LIN {X 0,Y 584.166,Z 578.172,A -85,B 0,C 180,E1 27168.047,E2 27168.047} C_VEL
LIN {X 0,Y 584.179,Z 576.67,A -85,B 0,C 180,E1 27167.893,E2 27167.893} C_VEL
LIN {X 0,Y 583.247,Z 571.34,A -85,B 0,C 180,E1 27167.345,E2 27167.345} C_VEL
LIN {X 0,Y 577.743,Z 558.263,A -85,B 0,C 180,E1 27166.095,E2 27166.095} C_VEL
LIN {X 0,Y 576.592,Z 552.276,A -85,B 0,C 180,E1 27165.618,E2 27165.618} C_VEL
LIN {X 0,Y 576.579,Z 551.371,A -85,B 0,C 180,E1 27165.553,E2 27165.553} C_VEL
LIN {X 0,Y 576.766,Z 536.079,A -85,B 0,C 180,E1 27164.583,E2 27164.583} C_VEL
LIN {X 0,Y 576.943,Z 519.51,A -85,B 0,C 180,E1 27163.761,E2 27163.761} C_VEL
LIN {X 0,Y 577.114,Z 502.31,A -85,B 0,C 180,E1 27163.13,E2 27163.13} C_VEL
LIN {X 0,Y 577.241,Z 485.032,A -85,B 0,C 180,E1 27162.689,E2 27162.689} C_VEL
LIN {X 0,Y 577.308,Z 459.491,A -85,B 0,C 180,E1 27162.321,E2 27162.321} C_VEL
LIN {X 0,Y 577.408,Z 315.564,A -85,B 0,C 180,E1 27160.474,E2 27160.474} C_VEL
LIN {X 0,Y 576.956,Z 312.588,A -85,B 0,C 180,E1 27160.407,E2 27160.407} C_VEL
LIN {X 0,Y 577.293,Z 276.085,A -85,B 0,C 180,E1 27157.226,E2 27157.226} C_VEL
LIN {X 0,Y 577.599,Z 242.251,A -85,B 0,C 180,E1 27154.246,E2 27154.246} C_VEL
LIN {X 0,Y 577.82,Z 208.346,A -85,B 0,C 180,E1 27151.246,E2 27151.246} C_VEL
LIN {X 0,Y 577.684,Z 175.567,A -85,B 0,C 180,E1 27148.382,E2 27148.382} C_VEL
LIN {X 0,Y 576.141,Z 169.97,A -85,B 0,C 180,E1 27147.806,E2 27147.806} C_VEL
LIN {X 0,Y 576.151,Z 169.971,A -85,B 0,C 180,E1 27144.48,E2 27144.48} C_VEL
LIN {X 0,Y 576.179,Z 170.097,A -85,B 0,C 180,E1 27141.143,E2 27141.143} C_VEL
LIN {X 0,Y 577.537,Z 173.559,A -85,B 0,C 180,E1 27141,E2 27141} C_VEL
LIN {X 0,Y 580.966,Z 179.3,A -85,B 0,C 180,E1 27140.689,E2 27140.689} C_VEL
LIN {X 0,Y 580.065,Z 404.117,A -85,B 0,C 180,E1 27137.526,E2 27137.526} C_VEL
LIN {X 0,Y 579.833,Z 463.496,A -85,B 0,C 180,E1 27136.673,E2 27136.673} C_VEL
LIN {X 0,Y 579.571,Z 484.812,A -85,B 0,C 180,E1 27136.178,E2 27136.178} C_VEL
LIN {X 0,Y 579.218,Z 506.984,A -85,B 0,C 180,E1 27135.474,E2 27135.474} C_VEL
LIN {X 0,Y 578.916,Z 528.199,A -85,B 0,C 180,E1 27134.601,E2 27134.601} C_VEL
LIN {X 0,Y 578.485,Z 549.01,A -85,B 0,C 180,E1 27133.533,E2 27133.533} C_VEL
LIN {X 0,Y 578.045,Z 569.167,A -85,B 0,C 180,E1 27132.289,E2 27132.289} C_VEL
LIN {X 0,Y 577.637,Z 588.568,A -85,B 0,C 180,E1 27130.867,E2 27130.867} C_VEL
LIN {X 0,Y 577.271,Z 606.408,A -85,B 0,C 180,E1 27129.341,E2 27129.341} C_VEL
LIN {X 0,Y 576.911,Z 623.556,A -85,B 0,C 180,E1 27127.623,E2 27127.623} C_VEL
LIN {X 0,Y 576.612,Z 638.899,A -85,B 0,C 180,E1 27125.836,E2 27125.836} C_VEL
LIN {X 0,Y 576.369,Z 652.746,A -85,B 0,C 180,E1 27123.959,E2 27123.959} C_VEL
LIN {X 0,Y 576.211,Z 664.765,A -85,B 0,C 180,E1 27122.072,E2 27122.072} C_VEL
LIN {X 0,Y 576.076,Z 675.919,A -85,B 0,C 180,E1 27119.991,E2 27119.991} C_VEL
LIN {X 0,Y 575.987,Z 685.052,A -85,B 0,C 180,E1 27117.922,E2 27117.922} C_VEL
LIN {X 0,Y 575.944,Z 692.576,A -85,B 0,C 180,E1 27115.833,E2 27115.833} C_VEL
LIN {X 0,Y 575.929,Z 698.241,A -85,B 0,C 180,E1 27113.805,E2 27113.805} C_VEL
LIN {X 0,Y 575.915,Z 702.695,A -85,B 0,C 180,E1 27111.596,E2 27111.596} C_VEL
LIN {X 0,Y 575.902,Z 705.381,A -85,B 0,C 180,E1 27109.472,E2 27109.472} C_VEL
LIN {X 0,Y 575.902,Z 706.413,A -85,B 0,C 180,E1 27107.375,E2 27107.375} C_VEL
LIN {X 0,Y 575.913,Z 705.871,A -85,B 0,C 180,E1 27105.139,E2 27105.139} C_VEL
LIN {X 0,Y 575.912,Z 703.824,A -85,B 0,C 180,E1 27103.044,E2 27103.044} C_VEL
LIN {X 0,Y 575.916,Z 700.064,A -85,B 0,C 180,E1 27100.908,E2 27100.908} C_VEL
LIN {X 0,Y 575.928,Z 694.42,A -85,B 0,C 180,E1 27098.687,E2 27098.687} C_VEL
LIN {X 0,Y 575.978,Z 687.766,A -85,B 0,C 180,E1 27096.679,E2 27096.679} C_VEL
LIN {X 0,Y 576.046,Z 679.006,A -85,B 0,C 180,E1 27094.58,E2 27094.58} C_VEL
LIN {X 0,Y 576.161,Z 668.424,A -85,B 0,C 180,E1 27092.487,E2 27092.487} C_VEL
LIN {X 0,Y 576.33,Z 656.46,A -85,B 0,C 180,E1 27090.497,E2 27090.497} C_VEL
LIN {X 0,Y 576.542,Z 643.064,A -85,B 0,C 180,E1 27088.609,E2 27088.609} C_VEL
LIN {X 0,Y 576.8,Z 628.359,A -85,B 0,C 180,E1 27086.82,E2 27086.82} C_VEL
LIN {X 0,Y 577.132,Z 611.742,A -85,B 0,C 180,E1 27085.081,E2 27085.081} C_VEL
LIN {X 0,Y 577.525,Z 594.068,A -85,B 0,C 180,E1 27083.489,E2 27083.489} C_VEL
LIN {X 0,Y 577.918,Z 576.003,A -85,B 0,C 180,E1 27082.094,E2 27082.094} C_VEL
LIN {X 0,Y 578.324,Z 556.324,A -85,B 0,C 180,E1 27080.803,E2 27080.803} C_VEL
LIN {X 0,Y 578.737,Z 535.219,A -85,B 0,C 180,E1 27079.649,E2 27079.649} C_VEL
LIN {X 0,Y 579.132,Z 515.257,A -85,B 0,C 180,E1 27078.75,E2 27078.75} C_VEL
LIN {X 0,Y 579.447,Z 493.278,A -85,B 0,C 180,E1 27077.974,E2 27077.974} C_VEL
LIN {X 0,Y 579.733,Z 471.198,A -85,B 0,C 180,E1 27077.398,E2 27077.398} C_VEL
LIN {X 0,Y 579.913,Z 449.201,A -85,B 0,C 180,E1 27077.008,E2 27077.008} C_VEL
LIN {X 0,Y 580.632,Z 243.532,A -85,B 0,C 180,E1 27074.13,E2 27074.13} C_VEL
LIN {X 0,Y 580.771,Z 178.82,A -85,B 0,C 180,E1 27073.202,E2 27073.202} C_VEL
LIN {X 0,Y 576.397,Z 171.192,A -85,B 0,C 180,E1 27072.798,E2 27072.798} C_VEL
LIN {X 0,Y 576.14,Z 169.971,A -85,B 0,C 180,E1 27072.737,E2 27072.737} C_VEL
LIN {X 0,Y 576.15,Z 169.971,A -85,B 0,C 180,E1 27069.479,E2 27069.479} C_VEL
LIN {X 0,Y 576.138,Z 169.966,A -85,B 0,C 180,E1 27066.258,E2 27066.258} C_VEL
LIN {X 0,Y 576.153,Z 169.963,A -85,B 0,C 180,E1 27062.956,E2 27062.956} C_VEL
LIN {X 0,Y 576.12,Z 169.969,A -85,B 0,C 180,E1 27059.667,E2 27059.667} C_VEL
LIN {X 0,Y 576.138,Z 169.97,A -85,B 0,C 180,E1 27056.411,E2 27056.411} C_VEL
LIN {X 0,Y 576.129,Z 169.971,A -85,B 0,C 180,E1 27053.136,E2 27053.136} C_VEL
LIN {X 0,Y 576.113,Z 169.969,A -85,B 0,C 180,E1 27049.918,E2 27049.918} C_VEL
LIN {X 0,Y 576.152,Z 169.964,A -85,B 0,C 180,E1 27046.647,E2 27046.647} C_VEL
LIN {X 0,Y 576.143,Z 169.967,A -85,B 0,C 180,E1 27043.352,E2 27043.352} C_VEL
LIN {X 0,Y 576.158,Z 169.967,A -85,B 0,C 180,E1 27040.066,E2 27040.066} C_VEL
LIN {X 0,Y 576.159,Z 169.965,A -85,B 0,C 180,E1 27036.703,E2 27036.703} C_VEL
LIN {X 0,Y 576.092,Z 169.971,A -85,B 0,C 180,E1 27033.499,E2 27033.499} C_VEL
LIN {X 0,Y 576.113,Z 169.968,A -85,B 0,C 180,E1 27030.104,E2 27030.104} C_VEL
LIN {X 0,Y 576.158,Z 169.964,A -85,B 0,C 180,E1 27026.876,E2 27026.876} C_VEL
LIN {X 0,Y 576.157,Z 169.966,A -85,B 0,C 180,E1 27023.525,E2 27023.525} C_VEL
LIN {X 0,Y 576.157,Z 169.967,A -85,B 0,C 180,E1 27020.203,E2 27020.203} C_VEL
LIN {X 0,Y 576.124,Z 169.965,A -85,B 0,C 180,E1 27017.009,E2 27017.009} C_VEL
LIN {X 0,Y 576.092,Z 169.967,A -85,B 0,C 180,E1 27013.756,E2 27013.756} C_VEL
LIN {X 0,Y 576.157,Z 169.967,A -85,B 0,C 180,E1 27010.6,E2 27010.6} C_VEL
LIN {X 0,Y 576.133,Z 169.968,A -85,B 0,C 180,E1 27007.379,E2 27007.379} C_VEL
LIN {X 0,Y 576.14,Z 169.962,A -85,B 0,C 180,E1 27004.081,E2 27004.081} C_VEL
LIN {X 0,Y 576.14,Z 169.964,A -85,B 0,C 180,E1 27000.895,E2 27000.895} C_VEL
LIN {X 0,Y 576.124,Z 169.969,A -85,B 0,C 180,E1 26997.514,E2 26997.514} C_VEL
LIN {X 0,Y 576.157,Z 169.969,A -85,B 0,C 180,E1 26994.323,E2 26994.323} C_VEL
LIN {X 0,Y 576.104,Z 169.969,A -85,B 0,C 180,E1 26991.115,E2 26991.115} C_VEL
LIN {X 0,Y 576.118,Z 169.965,A -85,B 0,C 180,E1 26987.878,E2 26987.878} C_VEL
LIN {X 0,Y 576.155,Z 169.964,A -85,B 0,C 180,E1 26984.706,E2 26984.706} C_VEL
LIN {X 0,Y 576.155,Z 169.968,A -85,B 0,C 180,E1 26981.357,E2 26981.357} C_VEL
LIN {X 0,Y 576.158,Z 169.964,A -85,B 0,C 180,E1 26978.093,E2 26978.093} C_VEL
LIN {X 0,Y 576.11,Z 169.969,A -85,B 0,C 180,E1 26974.946,E2 26974.946} C_VEL
LIN {X 0,Y 576.091,Z 169.971,A -85,B 0,C 180,E1 26971.605,E2 26971.605} C_VEL
LIN {X 0,Y 576.164,Z 169.967,A -85,B 0,C 180,E1 26968.51,E2 26968.51} C_VEL
LIN {X 0,Y 576.144,Z 169.97,A -85,B 0,C 180,E1 26965.171,E2 26965.171} C_VEL
LIN {X 0,Y 576.163,Z 170.139,A -85,B 0,C 180,E1 26963.964,E2 26963.964} C_VEL
LIN {X 0,Y 577.514,Z 173.558,A -85,B 0,C 180,E1 26963.57,E2 26963.57} C_VEL
LIN {X 0,Y 581.885,Z 182.987,A -85,B 0,C 180,E1 26962.442,E2 26962.442} C_VEL
LIN {X 0,Y 581.171,Z 223.856,A -85,B 0,C 180,E1 26959.435,E2 26959.435} C_VEL
LIN {X 0,Y 580.968,Z 264.821,A -85,B 0,C 180,E1 26956.496,E2 26956.496} C_VEL
LIN {X 0,Y 582.558,Z 275.609,A -85,B 0,C 180,E1 26955.621,E2 26955.621} C_VEL
LIN {X 0,Y 585.556,Z 284.297,A -85,B 0,C 180,E1 26954.808,E2 26954.808} C_VEL
LIN {X 0,Y 589.359,Z 290.159,A -85,B 0,C 180,E1 26954.141,E2 26954.141} C_VEL
LIN {X 0,Y 592.357,Z 293.003,A -85,B 0,C 180,E1 26953.604,E2 26953.604} C_VEL
LIN {X 0,Y 594.862,Z 294.195,A -85,B 0,C 180,E1 26953.017,E2 26953.017} C_VEL
LIN {X 0,Y 596.402,Z 293.842,A -85,B 0,C 180,E1 26952.469,E2 26952.469} C_VEL
LIN {X 0,Y 597.06,Z 292.212,A -85,B 0,C 180,E1 26951.927,E2 26951.927} C_VEL
LIN {X 0,Y 596.652,Z 289.094,A -85,B 0,C 180,E1 26951.383,E2 26951.383} C_VEL
LIN {X 0,Y 595.08,Z 284.676,A -85,B 0,C 180,E1 26950.925,E2 26950.925} C_VEL
LIN {X 0,Y 592.307,Z 278.496,A -85,B 0,C 180,E1 26950.559,E2 26950.559} C_VEL
LIN {X 0,Y 589.472,Z 269.594,A -85,B 0,C 180,E1 26950.235,E2 26950.235} C_VEL
LIN {X 0,Y 587.68,Z 259.22,A -85,B 0,C 180,E1 26950.028,E2 26950.028} C_VEL
LIN {X 0,Y 586.902,Z 246.138,A -85,B 0,C 180,E1 26949.938,E2 26949.938} C_VEL
LIN {X 0,Y 586.776,Z 183.916,A -85,B 0,C 180,E1 26949.923,E2 26949.923} C_VEL
LIN {X 0,Y 584.935,Z 181.56,A -85,B 0,C 180,E1 26949.707,E2 26949.707} C_VEL
LIN {X 0,Y 581.754,Z 178.104,A -85,B 0,C 180,E1 26949.329,E2 26949.329} C_VEL
LIN {X 0,Y 580.647,Z 176.215,A -85,B 0,C 180,E1 26949.195,E2 26949.195} C_VEL
LIN {X 0,Y 577.814,Z 173.937,A -85,B 0,C 180,E1 26948.849,E2 26948.849} C_VEL
LIN {X 0,Y 576.366,Z 171.038,A -85,B 0,C 180,E1 26948.67,E2 26948.67} C_VEL
LIN {X 0,Y 576.158,Z 169.97,A -85,B 0,C 180,E1 26948.627,E2 26948.627} C_VEL
LIN {X 0,Y 576.181,Z 170.151,A -85,B 0,C 180,E1 26948.44,E2 26948.44} C_VEL
LIN {X 0,Y 580.511,Z 180.927,A -85,B 0,C 180,E1 26947.321,E2 26947.321} C_VEL
LIN {X 0,Y 579.808,Z 224.835,A -85,B 0,C 180,E1 26944.266,E2 26944.266} C_VEL
LIN {X 0,Y 579.906,Z 227.325,A -85,B 0,C 180,E1 26944.125,E2 26944.125} C_VEL
LIN {X 0,Y 581.019,Z 234.139,A -85,B 0,C 180,E1 26943.951,E2 26943.951} C_VEL
LIN {X 0,Y 580.152,Z 452.345,A -85,B 0,C 180,E1 26940.873,E2 26940.873} C_VEL
LIN {X 0,Y 579.832,Z 532.96,A -85,B 0,C 180,E1 26939.727,E2 26939.727} C_VEL
LIN {X 0,Y 579.577,Z 555.095,A -85,B 0,C 180,E1 26939.217,E2 26939.217} C_VEL
LIN {X 0,Y 579.228,Z 577.783,A -85,B 0,C 180,E1 26938.49,E2 26938.49} C_VEL
LIN {X 0,Y 578.897,Z 598.757,A -85,B 0,C 180,E1 26937.62,E2 26937.62} C_VEL
LIN {X 0,Y 578.49,Z 618.753,A -85,B 0,C 180,E1 26936.593,E2 26936.593} C_VEL
LIN {X 0,Y 578.045,Z 638.958,A -85,B 0,C 180,E1 26935.347,E2 26935.347} C_VEL
LIN {X 0,Y 577.659,Z 658.111,A -85,B 0,C 180,E1 26933.95,E2 26933.95} C_VEL
LIN {X 0,Y 577.271,Z 676.271,A -85,B 0,C 180,E1 26932.399,E2 26932.399} C_VEL
LIN {X 0,Y 576.911,Z 693.951,A -85,B 0,C 180,E1 26930.629,E2 26930.629} C_VEL
LIN {X 0,Y 576.602,Z 709.761,A -85,B 0,C 180,E1 26928.775,E2 26928.775} C_VEL
LIN {X 0,Y 576.363,Z 723.17,A -85,B 0,C 180,E1 26926.944,E2 26926.944} C_VEL
LIN {X 0,Y 576.192,Z 735.515,A -85,B 0,C 180,E1 26924.984,E2 26924.984} C_VEL
LIN {X 0,Y 576.073,Z 746.408,A -85,B 0,C 180,E1 26922.938,E2 26922.938} C_VEL
LIN {X 0,Y 575.986,Z 755.302,A -85,B 0,C 180,E1 26920.907,E2 26920.907} C_VEL
LIN {X 0,Y 575.938,Z 762.863,A -85,B 0,C 180,E1 26918.788,E2 26918.788} C_VEL
LIN {X 0,Y 575.925,Z 768.682,A -85,B 0,C 180,E1 26916.68,E2 26916.68} C_VEL
LIN {X 0,Y 575.916,Z 772.79,A -85,B 0,C 180,E1 26914.58,E2 26914.58} C_VEL
LIN {X 0,Y 575.91,Z 775.488,A -85,B 0,C 180,E1 26912.388,E2 26912.388} C_VEL
LIN {X 0,Y 575.905,Z 776.473,A -85,B 0,C 180,E1 26910.199,E2 26910.199} C_VEL
LIN {X 0,Y 575.909,Z 775.822,A -85,B 0,C 180,E1 26908.109,E2 26908.109} C_VEL
LIN {X 0,Y 575.913,Z 773.582,A -85,B 0,C 180,E1 26905.918,E2 26905.918} C_VEL
LIN {X 0,Y 575.917,Z 769.79,A -85,B 0,C 180,E1 26903.821,E2 26903.821} C_VEL
LIN {X 0,Y 575.934,Z 764.368,A -85,B 0,C 180,E1 26901.711,E2 26901.711} C_VEL
LIN {X 0,Y 575.976,Z 757.695,A -85,B 0,C 180,E1 26899.7,E2 26899.7} C_VEL
LIN {X 0,Y 576.042,Z 749.224,A -85,B 0,C 180,E1 26897.672,E2 26897.672} C_VEL
LIN {X 0,Y 576.161,Z 738.987,A -85,B 0,C 180,E1 26895.631,E2 26895.631} C_VEL
LIN {X 0,Y 576.325,Z 727.346,A -85,B 0,C 180,E1 26893.677,E2 26893.677} C_VEL
LIN {X 0,Y 576.52,Z 714.246,A -85,B 0,C 180,E1 26891.809,E2 26891.809} C_VEL
LIN {X 0,Y 576.788,Z 698.895,A -85,B 0,C 180,E1 26889.926,E2 26889.926} C_VEL
LIN {X 0,Y 577.124,Z 682.718,A -85,B 0,C 180,E1 26888.219,E2 26888.219} C_VEL
LIN {X 0,Y 577.506,Z 665.385,A -85,B 0,C 180,E1 26886.642,E2 26886.642} C_VEL
LIN {X 0,Y 577.903,Z 646.751,A -85,B 0,C 180,E1 26885.193,E2 26885.193} C_VEL
LIN {X 0,Y 578.302,Z 627.096,A -85,B 0,C 180,E1 26883.895,E2 26883.895} C_VEL
LIN {X 0,Y 578.73,Z 606.41,A -85,B 0,C 180,E1 26882.752,E2 26882.752} C_VEL
LIN {X 0,Y 579.124,Z 585.901,A -85,B 0,C 180,E1 26881.823,E2 26881.823} C_VEL
LIN {X 0,Y 579.425,Z 564.416,A -85,B 0,C 180,E1 26881.056,E2 26881.056} C_VEL
LIN {X 0,Y 579.735,Z 542.303,A -85,B 0,C 180,E1 26880.466,E2 26880.466} C_VEL
LIN {X 0,Y 579.913,Z 520.195,A -85,B 0,C 180,E1 26880.067,E2 26880.067} C_VEL
LIN {X 0,Y 580.782,Z 292.439,A -85,B 0,C 180,E1 26876.88,E2 26876.88} C_VEL
LIN {X 0,Y 580.844,Z 228.358,A -85,B 0,C 180,E1 26875.953,E2 26875.953} C_VEL
LIN {X 0,Y 580.391,Z 224.044,A -85,B 0,C 180,E1 26875.832,E2 26875.832} C_VEL
LIN {X 0,Y 580.924,Z 180.697,A -85,B 0,C 180,E1 26873.742,E2 26873.742} C_VEL
LIN {X 0,Y 576.27,Z 170.651,A -85,B 0,C 180,E1 26872.894,E2 26872.894} C_VEL
LIN {X 0,Y 576.152,Z 169.971,A -85,B 0,C 180,E1 26872.848,E2 26872.848} C_VEL
LIN {X 0,Y 576.184,Z 170.204,A -85,B 0,C 180,E1 26871.352,E2 26871.352} C_VEL
LIN {X 0,Y 577.268,Z 173.153,A -85,B 0,C 180,E1 26871.218,E2 26871.218} C_VEL
LIN {X 0,Y 579.702,Z 175.67,A -85,B 0,C 180,E1 26870.92,E2 26870.92} C_VEL
LIN {X 0,Y 580.965,Z 176.724,A -85,B 0,C 180,E1 26870.766,E2 26870.766} C_VEL
LIN {X 0,Y 583.703,Z 180.482,A -85,B 0,C 180,E1 26870.438,E2 26870.438} C_VEL
LIN {X 0,Y 585.977,Z 182.712,A -85,B 0,C 180,E1 26870.17,E2 26870.17} C_VEL
LIN {X 0,Y 589.596,Z 186.957,A -85,B 0,C 180,E1 26869.75,E2 26869.75} C_VEL
LIN {X 0,Y 594.761,Z 192.611,A -85,B 0,C 180,E1 26869.159,E2 26869.159} C_VEL
LIN {X 0,Y 597.542,Z 195.032,A -85,B 0,C 180,E1 26868.691,E2 26868.691} C_VEL
LIN {X 0,Y 599.27,Z 196.446,A -85,B 0,C 180,E1 26868.134,E2 26868.134} C_VEL
LIN {X 0,Y 599.686,Z 197.232,A -85,B 0,C 180,E1 26867.613,E2 26867.613} C_VEL
LIN {X 0,Y 598.696,Z 198.051,A -85,B 0,C 180,E1 26867.011,E2 26867.011} C_VEL
LIN {X 0,Y 596.915,Z 197.512,A -85,B 0,C 180,E1 26866.493,E2 26866.493} C_VEL
LIN {X 0,Y 594.088,Z 195.403,A -85,B 0,C 180,E1 26865.943,E2 26865.943} C_VEL
LIN {X 0,Y 591.068,Z 193.123,A -85,B 0,C 180,E1 26865.55,E2 26865.55} C_VEL
LIN {X 0,Y 585.889,Z 188.609,A -85,B 0,C 180,E1 26864.952,E2 26864.952} C_VEL
LIN {X 0,Y 582.45,Z 183.25,A -85,B 0,C 180,E1 26864.428,E2 26864.428} C_VEL
LIN {X 0,Y 576.337,Z 170.931,A -85,B 0,C 180,E1 26863.324,E2 26863.324} C_VEL
LIN {X 0,Y 576.158,Z 169.971,A -85,B 0,C 180,E1 26863.241,E2 26863.241} C_VEL
LIN {X 0,Y 576.139,Z 169.964,A -85,B 0,C 180,E1 26859.949,E2 26859.949} C_VEL
LIN {X 0,Y 576.118,Z 169.969,A -85,B 0,C 180,E1 26856.656,E2 26856.656} C_VEL
LIN {X 0,Y 576.161,Z 169.969,A -85,B 0,C 180,E1 26853.413,E2 26853.413} C_VEL
LIN {X 0,Y 576.162,Z 170.086,A -85,B 0,C 180,E1 26851.16,E2 26851.16} C_VEL
LIN {X 0,Y 576.697,Z 174.6,A -85,B 0,C 180,E1 26850.819,E2 26850.819} C_VEL
LIN {X 0,Y 577.409,Z 207.54,A -85,B 0,C 180,E1 26848.324,E2 26848.324} C_VEL
LIN {X 0,Y 577.599,Z 237.816,A -85,B 0,C 180,E1 26845.863,E2 26845.863} C_VEL
LIN {X 0,Y 577.369,Z 272.172,A -85,B 0,C 180,E1 26842.932,E2 26842.932} C_VEL
LIN {X 0,Y 576.978,Z 310.15,A -85,B 0,C 180,E1 26839.697,E2 26839.697} C_VEL
LIN {X 0,Y 576.997,Z 313.03,A -85,B 0,C 180,E1 26839.483,E2 26839.483} C_VEL
LIN {X 0,Y 577.561,Z 319.15,A -85,B 0,C 180,E1 26839.384,E2 26839.384} C_VEL
LIN {X 0,Y 577.209,Z 481.726,A -85,B 0,C 180,E1 26837.282,E2 26837.282} C_VEL
LIN {X 0,Y 577.127,Z 499.279,A -85,B 0,C 180,E1 26836.872,E2 26836.872} C_VEL
LIN {X 0,Y 576.991,Z 515.78,A -85,B 0,C 180,E1 26836.303,E2 26836.303} C_VEL
LIN {X 0,Y 576.811,Z 532.277,A -85,B 0,C 180,E1 26835.534,E2 26835.534} C_VEL
LIN {X 0,Y 576.635,Z 547.335,A -85,B 0,C 180,E1 26834.636,E2 26834.636} C_VEL
LIN {X 0,Y 576.449,Z 562.025,A -85,B 0,C 180,E1 26833.542,E2 26833.542} C_VEL
LIN {X 0,Y 576.281,Z 575.839,A -85,B 0,C 180,E1 26832.271,E2 26832.271} C_VEL
LIN {X 0,Y 576.151,Z 587.921,A -85,B 0,C 180,E1 26830.903,E2 26830.903} C_VEL
LIN {X 0,Y 576.044,Z 598.713,A -85,B 0,C 180,E1 26829.39,E2 26829.39} C_VEL
LIN {X 0,Y 575.978,Z 607.856,A -85,B 0,C 180,E1 26827.782,E2 26827.782} C_VEL
LIN {X 0,Y 575.941,Z 614.944,A -85,B 0,C 180,E1 26826.179,E2 26826.179} C_VEL
LIN {X 0,Y 575.924,Z 620.472,A -85,B 0,C 180,E1 26824.48,E2 26824.48} C_VEL
LIN {X 0,Y 575.915,Z 624.302,A -85,B 0,C 180,E1 26822.686,E2 26822.686} C_VEL
LIN {X 0,Y 575.909,Z 626.225,A -85,B 0,C 180,E1 26820.895,E2 26820.895} C_VEL
LIN {X 0,Y 575.914,Z 626.333,A -85,B 0,C 180,E1 26819.204,E2 26819.204} C_VEL
LIN {X 0,Y 575.915,Z 624.602,A -85,B 0,C 180,E1 26817.412,E2 26817.412} C_VEL
LIN {X 0,Y 575.921,Z 620.948,A -85,B 0,C 180,E1 26815.619,E2 26815.619} C_VEL
LIN {X 0,Y 575.935,Z 615.645,A -85,B 0,C 180,E1 26813.921,E2 26813.921} C_VEL
LIN {X 0,Y 575.976,Z 608.813,A -85,B 0,C 180,E1 26812.318,E2 26812.318} C_VEL
LIN {X 0,Y 576.035,Z 599.922,A -85,B 0,C 180,E1 26810.71,E2 26810.71} C_VEL
LIN {X 0,Y 576.13,Z 589.382,A -85,B 0,C 180,E1 26809.197,E2 26809.197} C_VEL
LIN {X 0,Y 576.266,Z 577.477,A -85,B 0,C 180,E1 26807.809,E2 26807.809} C_VEL
LIN {X 0,Y 576.418,Z 564.288,A -85,B 0,C 180,E1 26806.559,E2 26806.559} C_VEL
LIN {X 0,Y 576.579,Z 551.371,A -85,B 0,C 180,E1 26805.553,E2 26805.553} C_VEL
LIN {X 0,Y 575.681,Z 545.123,A -85,B 0,C 180,E1 26805.102,E2 26805.102} C_VEL
LIN {X 0,Y 570.3,Z 530.053,A -85,B 0,C 180,E1 26804.075,E2 26804.075} C_VEL
LIN {X 0,Y 569.181,Z 522.294,A -85,B 0,C 180,E1 26803.662,E2 26803.662} C_VEL
LIN {X 0,Y 569.387,Z 506.325,A -85,B 0,C 180,E1 26803.026,E2 26803.026} C_VEL
LIN {X 0,Y 569.555,Z 489.29,A -85,B 0,C 180,E1 26802.544,E2 26802.544} C_VEL
LIN {X 0,Y 569.665,Z 470.385,A -85,B 0,C 180,E1 26802.217,E2 26802.217} C_VEL
LIN {X 0,Y 569.852,Z 316.495,A -85,B 0,C 180,E1 26800.217,E2 26800.217} C_VEL
LIN {X 0,Y 569.247,Z 312.464,A -85,B 0,C 180,E1 26800.12,E2 26800.12} C_VEL
LIN {X 0,Y 569.705,Z 277.5,A -85,B 0,C 180,E1 26797.014,E2 26797.014} C_VEL
LIN {X 0,Y 570.079,Z 241.888,A -85,B 0,C 180,E1 26793.851,E2 26793.851} C_VEL
LIN {X 0,Y 570.312,Z 209.094,A -85,B 0,C 180,E1 26790.946,E2 26790.946} C_VEL
LIN {X 0,Y 570.279,Z 178.323,A -85,B 0,C 180,E1 26788.249,E2 26788.249} C_VEL
LIN {X 0,Y 568.213,Z 170.957,A -85,B 0,C 180,E1 26787.491,E2 26787.491} C_VEL
LIN {X 0,Y 568.193,Z 170.959,A -85,B 0,C 180,E1 26784.127,E2 26784.127} C_VEL
LIN {X 0,Y 568.211,Z 171.117,A -85,B 0,C 180,E1 26781.675,E2 26781.675} C_VEL
LIN {X 0,Y 569.487,Z 174.414,A -85,B 0,C 180,E1 26781.537,E2 26781.537} C_VEL
LIN {X 0,Y 571.236,Z 177.159,A -85,B 0,C 180,E1 26781.375,E2 26781.375} C_VEL
LIN {X 0,Y 574.293,Z 182.62,A -85,B 0,C 180,E1 26781.085,E2 26781.085} C_VEL
LIN {X 0,Y 573.165,Z 406.563,A -85,B 0,C 180,E1 26777.899,E2 26777.899} C_VEL
LIN {X 0,Y 572.876,Z 463.7,A -85,B 0,C 180,E1 26777.067,E2 26777.067} C_VEL
LIN {X 0,Y 572.549,Z 485.027,A -85,B 0,C 180,E1 26776.566,E2 26776.566} C_VEL
LIN {X 0,Y 572.135,Z 506.682,A -85,B 0,C 180,E1 26775.872,E2 26775.872} C_VEL
LIN {X 0,Y 571.735,Z 527.721,A -85,B 0,C 180,E1 26775.001,E2 26775.001} C_VEL
LIN {X 0,Y 571.185,Z 548.622,A -85,B 0,C 180,E1 26773.922,E2 26773.922} C_VEL
LIN {X 0,Y 570.668,Z 568.42,A -85,B 0,C 180,E1 26772.692,E2 26772.692} C_VEL
LIN {X 0,Y 570.164,Z 587.116,A -85,B 0,C 180,E1 26771.319,E2 26771.319} C_VEL
LIN {X 0,Y 569.683,Z 604.411,A -85,B 0,C 180,E1 26769.838,E2 26769.838} C_VEL
LIN {X 0,Y 569.224,Z 621.861,A -85,B 0,C 180,E1 26768.1,E2 26768.1} C_VEL
LIN {X 0,Y 568.85,Z 637.152,A -85,B 0,C 180,E1 26766.324,E2 26766.324} C_VEL
LIN {X 0,Y 568.536,Z 652.019,A -85,B 0,C 180,E1 26764.309,E2 26764.309} C_VEL
LIN {X 0,Y 568.321,Z 664.211,A -85,B 0,C 180,E1 26762.384,E2 26762.384} C_VEL
LIN {X 0,Y 568.134,Z 675.718,A -85,B 0,C 180,E1 26760.218,E2 26760.218} C_VEL
LIN {X 0,Y 568.021,Z 684.855,A -85,B 0,C 180,E1 26758.128,E2 26758.128} C_VEL
LIN {X 0,Y 567.963,Z 692.456,A -85,B 0,C 180,E1 26755.999,E2 26755.999} C_VEL
LIN {X 0,Y 567.933,Z 698.282,A -85,B 0,C 180,E1 26753.886,E2 26753.886} C_VEL
LIN {X 0,Y 567.914,Z 702.641,A -85,B 0,C 180,E1 26751.699,E2 26751.699} C_VEL
LIN {X 0,Y 567.901,Z 705.349,A -85,B 0,C 180,E1 26749.543,E2 26749.543} C_VEL
LIN {X 0,Y 567.902,Z 706.41,A -85,B 0,C 180,E1 26747.396,E2 26747.396} C_VEL
LIN {X 0,Y 567.915,Z 705.866,A -85,B 0,C 180,E1 26745.104,E2 26745.104} C_VEL
LIN {X 0,Y 567.91,Z 703.73,A -85,B 0,C 180,E1 26742.921,E2 26742.921} C_VEL
LIN {X 0,Y 567.911,Z 699.931,A -85,B 0,C 180,E1 26740.756,E2 26740.756} C_VEL
LIN {X 0,Y 567.934,Z 694.528,A -85,B 0,C 180,E1 26738.606,E2 26738.606} C_VEL
LIN {X 0,Y 567.993,Z 687.895,A -85,B 0,C 180,E1 26736.57,E2 26736.57} C_VEL
LIN {X 0,Y 568.081,Z 679.181,A -85,B 0,C 180,E1 26734.442,E2 26734.442} C_VEL
LIN {X 0,Y 568.226,Z 668.647,A -85,B 0,C 180,E1 26732.32,E2 26732.32} C_VEL
LIN {X 0,Y 568.441,Z 656.726,A -85,B 0,C 180,E1 26730.303,E2 26730.303} C_VEL
LIN {X 0,Y 568.716,Z 643.363,A -85,B 0,C 180,E1 26728.388,E2 26728.388} C_VEL
LIN {X 0,Y 569.054,Z 628.72,A -85,B 0,C 180,E1 26726.575,E2 26726.575} C_VEL
LIN {X 0,Y 569.476,Z 612.164,A -85,B 0,C 180,E1 26724.812,E2 26724.812} C_VEL
LIN {X 0,Y 569.949,Z 595.181,A -85,B 0,C 180,E1 26723.25,E2 26723.25} C_VEL
LIN {X 0,Y 570.447,Z 576.852,A -85,B 0,C 180,E1 26721.81,E2 26721.81} C_VEL
LIN {X 0,Y 570.951,Z 557.704,A -85,B 0,C 180,E1 26720.525,E2 26720.525} C_VEL
LIN {X 0,Y 571.458,Z 537.985,A -85,B 0,C 180,E1 26719.414,E2 26719.414} C_VEL
LIN {X 0,Y 571.899,Z 518.451,A -85,B 0,C 180,E1 26718.504,E2 26718.504} C_VEL
LIN {X 0,Y 572.34,Z 496.753,A -85,B 0,C 180,E1 26717.694,E2 26717.694} C_VEL
LIN {X 0,Y 572.729,Z 474.998,A -85,B 0,C 180,E1 26717.085,E2 26717.085} C_VEL
LIN {X 0,Y 572.93,Z 453.631,A -85,B 0,C 180,E1 26716.675,E2 26716.675} C_VEL
LIN {X 0,Y 573.884,Z 247.929,A -85,B 0,C 180,E1 26713.759,E2 26713.759} C_VEL
LIN {X 0,Y 574.094,Z 182.048,A -85,B 0,C 180,E1 26712.803,E2 26712.803} C_VEL
LIN {X 0,Y 569.856,Z 174.958,A -85,B 0,C 180,E1 26712.407,E2 26712.407} C_VEL
LIN {X 0,Y 568.271,Z 171.594,A -85,B 0,C 180,E1 26712.246,E2 26712.246} C_VEL
LIN {X 0,Y 568.165,Z 170.961,A -85,B 0,C 180,E1 26712.217,E2 26712.217} C_VEL
LIN {X 0,Y 568.223,Z 170.956,A -85,B 0,C 180,E1 26709.072,E2 26709.072} C_VEL
LIN {X 0,Y 568.218,Z 170.959,A -85,B 0,C 180,E1 26705.685,E2 26705.685} C_VEL
LIN {X 0,Y 568.216,Z 170.957,A -85,B 0,C 180,E1 26702.319,E2 26702.319} C_VEL
LIN {X 0,Y 568.197,Z 170.956,A -85,B 0,C 180,E1 26699.081,E2 26699.081} C_VEL
LIN {X 0,Y 568.156,Z 170.958,A -85,B 0,C 180,E1 26695.805,E2 26695.805} C_VEL
LIN {X 0,Y 568.189,Z 170.955,A -85,B 0,C 180,E1 26692.528,E2 26692.528} C_VEL
LIN {X 0,Y 568.215,Z 170.959,A -85,B 0,C 180,E1 26689.325,E2 26689.325} C_VEL
LIN {X 0,Y 568.198,Z 170.957,A -85,B 0,C 180,E1 26686.032,E2 26686.032} C_VEL
LIN {X 0,Y 568.217,Z 170.952,A -85,B 0,C 180,E1 26682.646,E2 26682.646} C_VEL
LIN {X 0,Y 568.183,Z 170.956,A -85,B 0,C 180,E1 26679.418,E2 26679.418} C_VEL
LIN {X 0,Y 568.185,Z 170.958,A -85,B 0,C 180,E1 26676.123,E2 26676.123} C_VEL
LIN {X 0,Y 568.199,Z 170.96,A -85,B 0,C 180,E1 26672.926,E2 26672.926} C_VEL
LIN {X 0,Y 568.171,Z 170.958,A -85,B 0,C 180,E1 26669.753,E2 26669.753} C_VEL
LIN {X 0,Y 568.214,Z 170.951,A -85,B 0,C 180,E1 26666.549,E2 26666.549} C_VEL
LIN {X 0,Y 568.205,Z 170.951,A -85,B 0,C 180,E1 26663.215,E2 26663.215} C_VEL
LIN {X 0,Y 568.217,Z 170.959,A -85,B 0,C 180,E1 26659.961,E2 26659.961} C_VEL
LIN {X 0,Y 568.212,Z 170.953,A -85,B 0,C 180,E1 26656.668,E2 26656.668} C_VEL
LIN {X 0,Y 568.149,Z 170.956,A -85,B 0,C 180,E1 26653.537,E2 26653.537} C_VEL
LIN {X 0,Y 568.197,Z 170.955,A -85,B 0,C 180,E1 26650.34,E2 26650.34} C_VEL
LIN {X 0,Y 568.225,Z 170.958,A -85,B 0,C 180,E1 26647.057,E2 26647.057} C_VEL
LIN {X 0,Y 568.207,Z 170.953,A -85,B 0,C 180,E1 26643.733,E2 26643.733} C_VEL
LIN {X 0,Y 568.22,Z 170.951,A -85,B 0,C 180,E1 26640.404,E2 26640.404} C_VEL
LIN {X 0,Y 568.177,Z 170.956,A -85,B 0,C 180,E1 26637.176,E2 26637.176} C_VEL
LIN {X 0,Y 568.171,Z 170.96,A -85,B 0,C 180,E1 26633.868,E2 26633.868} C_VEL
LIN {X 0,Y 568.21,Z 170.958,A -85,B 0,C 180,E1 26630.684,E2 26630.684} C_VEL
LIN {X 0,Y 568.186,Z 170.956,A -85,B 0,C 180,E1 26627.397,E2 26627.397} C_VEL
LIN {X 0,Y 568.202,Z 170.953,A -85,B 0,C 180,E1 26624.067,E2 26624.067} C_VEL
LIN {X 0,Y 568.203,Z 170.955,A -85,B 0,C 180,E1 26620.789,E2 26620.789} C_VEL
LIN {X 0,Y 568.192,Z 170.959,A -85,B 0,C 180,E1 26617.442,E2 26617.442} C_VEL
LIN {X 0,Y 568.223,Z 170.959,A -85,B 0,C 180,E1 26614.239,E2 26614.239} C_VEL
LIN {X 0,Y 568.167,Z 170.96,A -85,B 0,C 180,E1 26610.942,E2 26610.942} C_VEL
LIN {X 0,Y 568.175,Z 170.961,A -85,B 0,C 180,E1 26607.639,E2 26607.639} C_VEL
LIN {X 0,Y 568.218,Z 170.964,A -85,B 0,C 180,E1 26604.66,E2 26604.66} C_VEL
LIN {X 0,Y 569.643,Z 174.611,A -85,B 0,C 180,E1 26604.233,E2 26604.233} C_VEL
LIN {X 0,Y 575.394,Z 186.846,A -85,B 0,C 180,E1 26602.737,E2 26602.737} C_VEL
LIN {X 0,Y 574.517,Z 227.602,A -85,B 0,C 180,E1 26599.713,E2 26599.713} C_VEL
LIN {X 0,Y 574.164,Z 267.554,A -85,B 0,C 180,E1 26596.814,E2 26596.814} C_VEL
LIN {X 0,Y 575.799,Z 279.097,A -85,B 0,C 180,E1 26595.867,E2 26595.867} C_VEL
LIN {X 0,Y 578.917,Z 288.411,A -85,B 0,C 180,E1 26594.988,E2 26594.988} C_VEL
LIN {X 0,Y 582.683,Z 294.598,A -85,B 0,C 180,E1 26594.298,E2 26594.298} C_VEL
LIN {X 0,Y 587.242,Z 299.166,A -85,B 0,C 180,E1 26593.646,E2 26593.646} C_VEL
LIN {X 0,Y 590.318,Z 300.962,A -85,B 0,C 180,E1 26593.113,E2 26593.113} C_VEL
LIN {X 0,Y 592.765,Z 301.296,A -85,B 0,C 180,E1 26592.514,E2 26592.514} C_VEL
LIN {X 0,Y 594.139,Z 300.148,A -85,B 0,C 180,E1 26591.92,E2 26591.92} C_VEL
LIN {X 0,Y 594.316,Z 297.612,A -85,B 0,C 180,E1 26591.331,E2 26591.331} C_VEL
LIN {X 0,Y 593.247,Z 293.902,A -85,B 0,C 180,E1 26590.822,E2 26590.822} C_VEL
LIN {X 0,Y 591.037,Z 289.251,A -85,B 0,C 180,E1 26590.417,E2 26590.417} C_VEL
LIN {X 0,Y 587.259,Z 281.029,A -85,B 0,C 180,E1 26589.979,E2 26589.979} C_VEL
LIN {X 0,Y 584.417,Z 271.352,A -85,B 0,C 180,E1 26589.646,E2 26589.646} C_VEL
LIN {X 0,Y 582.587,Z 260.103,A -85,B 0,C 180,E1 26589.428,E2 26589.428} C_VEL
LIN {X 0,Y 581.802,Z 246.434,A -85,B 0,C 180,E1 26589.334,E2 26589.334} C_VEL
LIN {X 0,Y 581.754,Z 187.971,A -85,B 0,C 180,E1 26589.329,E2 26589.329} C_VEL
LIN {X 0,Y 578.128,Z 183.671,A -85,B 0,C 180,E1 26588.888,E2 26588.888} C_VEL
LIN {X 0,Y 574.536,Z 180.188,A -85,B 0,C 180,E1 26588.442,E2 26588.442} C_VEL
LIN {X 0,Y 572.522,Z 180.259,A -85,B 0,C 180,E1 26588.187,E2 26588.187} C_VEL
LIN {X 0,Y 571.743,Z 179.782,A -85,B 0,C 180,E1 26588.078,E2 26588.078} C_VEL
LIN {X 0,Y 573.683,Z 184.371,A -85,B 0,C 180,E1 26587.59,E2 26587.59} C_VEL
LIN {X 0,Y 572.909,Z 227.019,A -85,B 0,C 180,E1 26584.605,E2 26584.605} C_VEL
LIN {X 0,Y 574.375,Z 235.64,A -85,B 0,C 180,E1 26584.376,E2 26584.376} C_VEL
LIN {X 0,Y 573.274,Z 454.189,A -85,B 0,C 180,E1 26581.259,E2 26581.259} C_VEL
LIN {X 0,Y 572.877,Z 532.947,A -85,B 0,C 180,E1 26580.125,E2 26580.125} C_VEL
LIN {X 0,Y 572.556,Z 555.224,A -85,B 0,C 180,E1 26579.608,E2 26579.608} C_VEL
LIN {X 0,Y 572.139,Z 577.376,A -85,B 0,C 180,E1 26578.892,E2 26578.892} C_VEL
LIN {X 0,Y 571.707,Z 598.694,A -85,B 0,C 180,E1 26578.001,E2 26578.001} C_VEL
LIN {X 0,Y 571.187,Z 618.761,A -85,B 0,C 180,E1 26576.961,E2 26576.961} C_VEL
LIN {X 0,Y 570.673,Z 638.161,A -85,B 0,C 180,E1 26575.754,E2 26575.754} C_VEL
LIN {X 0,Y 570.182,Z 656.802,A -85,B 0,C 180,E1 26574.391,E2 26574.391} C_VEL
LIN {X 0,Y 569.662,Z 675.694,A -85,B 0,C 180,E1 26572.769,E2 26572.769} C_VEL
LIN {X 0,Y 569.199,Z 692.732,A -85,B 0,C 180,E1 26571.053,E2 26571.053} C_VEL
LIN {X 0,Y 568.838,Z 707.829,A -85,B 0,C 180,E1 26569.284,E2 26569.284} C_VEL
LIN {X 0,Y 568.545,Z 721.759,A -85,B 0,C 180,E1 26567.395,E2 26567.395} C_VEL
LIN {X 0,Y 568.31,Z 734.412,A -85,B 0,C 180,E1 26565.394,E2 26565.394} C_VEL
LIN {X 0,Y 568.139,Z 745.381,A -85,B 0,C 180,E1 26563.329,E2 26563.329} C_VEL
LIN {X 0,Y 568.022,Z 754.898,A -85,B 0,C 180,E1 26561.164,E2 26561.164} C_VEL
LIN {X 0,Y 567.965,Z 762.563,A -85,B 0,C 180,E1 26559.014,E2 26559.014} C_VEL
LIN {X 0,Y 567.933,Z 768.577,A -85,B 0,C 180,E1 26556.817,E2 26556.817} C_VEL
LIN {X 0,Y 567.918,Z 772.793,A -85,B 0,C 180,E1 26554.645,E2 26554.645} C_VEL
LIN {X 0,Y 567.909,Z 775.489,A -85,B 0,C 180,E1 26552.422,E2 26552.422} C_VEL
LIN {X 0,Y 567.905,Z 776.475,A -85,B 0,C 180,E1 26550.202,E2 26550.202} C_VEL
LIN {X 0,Y 567.912,Z 775.758,A -85,B 0,C 180,E1 26547.982,E2 26547.982} C_VEL
LIN {X 0,Y 567.911,Z 773.427,A -85,B 0,C 180,E1 26545.759,E2 26545.759} C_VEL
LIN {X 0,Y 567.916,Z 769.586,A -85,B 0,C 180,E1 26543.632,E2 26543.632} C_VEL
LIN {X 0,Y 567.936,Z 764.08,A -85,B 0,C 180,E1 26541.496,E2 26541.496} C_VEL
LIN {X 0,Y 567.995,Z 756.926,A -85,B 0,C 180,E1 26539.348,E2 26539.348} C_VEL
LIN {X 0,Y 568.088,Z 748.302,A -85,B 0,C 180,E1 26537.29,E2 26537.29} C_VEL
LIN {X 0,Y 568.231,Z 737.833,A -85,B 0,C 180,E1 26535.218,E2 26535.218} C_VEL
LIN {X 0,Y 568.452,Z 725.998,A -85,B 0,C 180,E1 26533.234,E2 26533.234} C_VEL
LIN {X 0,Y 568.756,Z 711.904,A -85,B 0,C 180,E1 26531.233,E2 26531.233} C_VEL
LIN {X 0,Y 569.105,Z 697.042,A -85,B 0,C 180,E1 26529.428,E2 26529.428} C_VEL
LIN {X 0,Y 569.526,Z 680.535,A -85,B 0,C 180,E1 26527.698,E2 26527.698} C_VEL
LIN {X 0,Y 569.996,Z 662.779,A -85,B 0,C 180,E1 26526.096,E2 26526.096} C_VEL
LIN {X 0,Y 570.521,Z 644.526,A -85,B 0,C 180,E1 26524.683,E2 26524.683} C_VEL
LIN {X 0,Y 571.061,Z 624.434,A -85,B 0,C 180,E1 26523.37,E2 26523.37} C_VEL
LIN {X 0,Y 571.529,Z 604.179,A -85,B 0,C 180,E1 26522.267,E2 26522.267} C_VEL
LIN {X 0,Y 572.047,Z 583.28,A -85,B 0,C 180,E1 26521.333,E2 26521.333} C_VEL
LIN {X 0,Y 572.454,Z 561.668,A -85,B 0,C 180,E1 26520.578,E2 26520.578} C_VEL
LIN {X 0,Y 572.77,Z 540.004,A -85,B 0,C 180,E1 26520.019,E2 26520.019} C_VEL
LIN {X 0,Y 573.001,Z 515.741,A -85,B 0,C 180,E1 26519.605,E2 26519.605} C_VEL
LIN {X 0,Y 574.094,Z 289.131,A -85,B 0,C 180,E1 26516.395,E2 26516.395} C_VEL
LIN {X 0,Y 574.203,Z 229.592,A -85,B 0,C 180,E1 26515.522,E2 26515.522} C_VEL
LIN {X 0,Y 573.604,Z 223.837,A -85,B 0,C 180,E1 26515.361,E2 26515.361} C_VEL
LIN {X 0,Y 574.113,Z 183.916,A -85,B 0,C 180,E1 26513.404,E2 26513.404} C_VEL
LIN {X 0,Y 569.318,Z 174.154,A -85,B 0,C 180,E1 26512.544,E2 26512.544} C_VEL
LIN {X 0,Y 568.414,Z 172.065,A -85,B 0,C 180,E1 26512.343,E2 26512.343} C_VEL
LIN {X 0,Y 569.906,Z 174.983,A -85,B 0,C 180,E1 26512.149,E2 26512.149} C_VEL
LIN {X 0,Y 572.832,Z 177.241,A -85,B 0,C 180,E1 26511.773,E2 26511.773} C_VEL
LIN {X 0,Y 575.783,Z 181.416,A -85,B 0,C 180,E1 26511.402,E2 26511.402} C_VEL
LIN {X 0,Y 578.208,Z 183.779,A -85,B 0,C 180,E1 26511.102,E2 26511.102} C_VEL
LIN {X 0,Y 581.756,Z 187.961,A -85,B 0,C 180,E1 26510.671,E2 26510.671} C_VEL
LIN {X 0,Y 591.863,Z 199.262,A -85,B 0,C 180,E1 26509.492,E2 26509.492} C_VEL
LIN {X 0,Y 594.914,Z 201.896,A -85,B 0,C 180,E1 26509.045,E2 26509.045} C_VEL
LIN {X 0,Y 596.981,Z 203.733,A -85,B 0,C 180,E1 26508.474,E2 26508.474} C_VEL
LIN {X 0,Y 597.659,Z 204.646,A -85,B 0,C 180,E1 26507.827,E2 26507.827} C_VEL
LIN {X 0,Y 596.61,Z 205.594,A -85,B 0,C 180,E1 26507.226,E2 26507.226} C_VEL
LIN {X 0,Y 594.296,Z 205.116,A -85,B 0,C 180,E1 26506.619,E2 26506.619} C_VEL
LIN {X 0,Y 591.192,Z 203.267,A -85,B 0,C 180,E1 26506.094,E2 26506.094} C_VEL
LIN {X 0,Y 586.722,Z 199.838,A -85,B 0,C 180,E1 26505.564,E2 26505.564} C_VEL
LIN {X 0,Y 581.489,Z 195.504,A -85,B 0,C 180,E1 26504.967,E2 26504.967} C_VEL
LIN {X 0,Y 577.456,Z 190.033,A -85,B 0,C 180,E1 26504.388,E2 26504.388} C_VEL
LIN {X 0,Y 569.443,Z 174.339,A -85,B 0,C 180,E1 26502.943,E2 26502.943} C_VEL
LIN {X 0,Y 568.188,Z 170.96,A -85,B 0,C 180,E1 26502.644,E2 26502.644} C_VEL
LIN {X 0,Y 568.22,Z 170.957,A -85,B 0,C 180,E1 26499.422,E2 26499.422} C_VEL
LIN {X 0,Y 568.179,Z 170.956,A -85,B 0,C 180,E1 26496.248,E2 26496.248} C_VEL
LIN {X 0,Y 568.189,Z 170.961,A -85,B 0,C 180,E1 26492.924,E2 26492.924} C_VEL
LIN {X 0,Y 568.233,Z 171.044,A -85,B 0,C 180,E1 26491.329,E2 26491.329} C_VEL
LIN {X 0,Y 568.949,Z 176.139,A -85,B 0,C 180,E1 26490.951,E2 26490.951} C_VEL
LIN {X 0,Y 569.603,Z 204.426,A -85,B 0,C 180,E1 26488.845,E2 26488.845} C_VEL
LIN {X 0,Y 569.975,Z 236.178,A -85,B 0,C 180,E1 26486.31,E2 26486.31} C_VEL
LIN {X 0,Y 569.855,Z 270.569,A -85,B 0,C 180,E1 26483.415,E2 26483.415} C_VEL
LIN {X 0,Y 569.317,Z 308.913,A -85,B 0,C 180,E1 26480.08,E2 26480.08} C_VEL
LIN {X 0,Y 569.294,Z 312.994,A -85,B 0,C 180,E1 26479.759,E2 26479.759} C_VEL
LIN {X 0,Y 570.016,Z 319.718,A -85,B 0,C 180,E1 26479.645,E2 26479.645} C_VEL
LIN {X 0,Y 569.568,Z 481.714,A -85,B 0,C 180,E1 26477.521,E2 26477.521} C_VEL
LIN {X 0,Y 569.459,Z 499.083,A -85,B 0,C 180,E1 26477.113,E2 26477.113} C_VEL
LIN {X 0,Y 569.283,Z 515.809,A -85,B 0,C 180,E1 26476.53,E2 26476.53} C_VEL
LIN {X 0,Y 569.055,Z 532.288,A -85,B 0,C 180,E1 26475.751,E2 26475.751} C_VEL
LIN {X 0,Y 568.822,Z 547.796,A -85,B 0,C 180,E1 26474.81,E2 26474.81} C_VEL
LIN {X 0,Y 568.6,Z 562.036,A -85,B 0,C 180,E1 26473.732,E2 26473.732} C_VEL
LIN {X 0,Y 568.385,Z 575.85,A -85,B 0,C 180,E1 26472.444,E2 26472.444} C_VEL
LIN {X 0,Y 568.215,Z 587.923,A -85,B 0,C 180,E1 26471.058,E2 26471.058} C_VEL
LIN {X 0,Y 568.084,Z 598.721,A -85,B 0,C 180,E1 26469.523,E2 26469.523} C_VEL
LIN {X 0,Y 567.995,Z 607.857,A -85,B 0,C 180,E1 26467.892,E2 26467.892} C_VEL
LIN {X 0,Y 567.948,Z 614.945,A -85,B 0,C 180,E1 26466.266,E2 26466.266} C_VEL
LIN {X 0,Y 567.927,Z 620.476,A -85,B 0,C 180,E1 26464.544,E2 26464.544} C_VEL
LIN {X 0,Y 567.915,Z 624.306,A -85,B 0,C 180,E1 26462.724,E2 26462.724} C_VEL
LIN {X 0,Y 567.909,Z 626.224,A -85,B 0,C 180,E1 26460.908,E2 26460.908} C_VEL
LIN {X 0,Y 567.913,Z 626.331,A -85,B 0,C 180,E1 26459.193,E2 26459.193} C_VEL
LIN {X 0,Y 567.915,Z 624.605,A -85,B 0,C 180,E1 26457.376,E2 26457.376} C_VEL
LIN {X 0,Y 567.922,Z 620.948,A -85,B 0,C 180,E1 26455.557,E2 26455.557} C_VEL
LIN {X 0,Y 567.943,Z 615.64,A -85,B 0,C 180,E1 26453.835,E2 26453.835} C_VEL
LIN {X 0,Y 567.992,Z 608.81,A -85,B 0,C 180,E1 26452.209,E2 26452.209} C_VEL
LIN {X 0,Y 568.069,Z 599.923,A -85,B 0,C 180,E1 26450.579,E2 26450.579} C_VEL
LIN {X 0,Y 568.194,Z 589.379,A -85,B 0,C 180,E1 26449.044,E2 26449.044} C_VEL
LIN {X 0,Y 568.355,Z 578.154,A -85,B 0,C 180,E1 26447.709,E2 26447.709} C_VEL
LIN {X 0,Y 568.552,Z 564.887,A -85,B 0,C 180,E1 26446.421,E2 26446.421} C_VEL
LIN {X 0,Y 568.796,Z 549.721,A -85,B 0,C 180,E1 26445.233,E2 26445.233} C_VEL
LIN {X 0,Y 569.02,Z 534.854,A -85,B 0,C 180,E1 26444.299,E2 26444.299} C_VEL
LIN {X 0,Y 569.181,Z 522.294,A -85,B 0,C 180,E1 26443.662,E2 26443.662} C_VEL
LIN {X 0,Y 568.322,Z 515.311,A -85,B 0,C 180,E1 26443.329,E2 26443.329} C_VEL
LIN {X 0,Y 562.995,Z 498.622,A -85,B 0,C 180,E1 26442.581,E2 26442.581} C_VEL
LIN {X 0,Y 561.914,Z 491.303,A -85,B 0,C 180,E1 26442.349,E2 26442.349} C_VEL
LIN {X 0,Y 561.899,Z 490.227,A -85,B 0,C 180,E1 26442.322,E2 26442.322} C_VEL
LIN {X 0,Y 562.044,Z 471.082,A -85,B 0,C 180,E1 26441.978,E2 26441.978} C_VEL
LIN {X 0,Y 562.315,Z 317.517,A -85,B 0,C 180,E1 26439.956,E2 26439.956} C_VEL
LIN {X 0,Y 561.564,Z 312.664,A -85,B 0,C 180,E1 26439.847,E2 26439.847} C_VEL
LIN {X 0,Y 562.176,Z 276.726,A -85,B 0,C 180,E1 26436.598,E2 26436.598} C_VEL
LIN {X 0,Y 562.562,Z 240.671,A -85,B 0,C 180,E1 26433.381,E2 26433.381} C_VEL
LIN {X 0,Y 562.79,Z 207.737,A -85,B 0,C 180,E1 26430.461,E2 26430.461} C_VEL
LIN {X 0,Y 562.643,Z 180.204,A -85,B 0,C 180,E1 26428.023,E2 26428.023} C_VEL
LIN {X 0,Y 560.279,Z 171.947,A -85,B 0,C 180,E1 26427.145,E2 26427.145} C_VEL
LIN {X 0,Y 560.252,Z 171.948,A -85,B 0,C 180,E1 26423.918,E2 26423.918} C_VEL
LIN {X 0,Y 560.275,Z 172.144,A -85,B 0,C 180,E1 26422.224,E2 26422.224} C_VEL
LIN {X 0,Y 561.631,Z 175.55,A -85,B 0,C 180,E1 26422.074,E2 26422.074} C_VEL
LIN {X 0,Y 563.295,Z 178.133,A -85,B 0,C 180,E1 26421.915,E2 26421.915} C_VEL
LIN {X 0,Y 567.651,Z 185.65,A -85,B 0,C 180,E1 26421.495,E2 26421.495} C_VEL
LIN {X 0,Y 566.288,Z 409.206,A -85,B 0,C 180,E1 26418.279,E2 26418.279} C_VEL
LIN {X 0,Y 565.946,Z 463.83,A -85,B 0,C 180,E1 26417.471,E2 26417.471} C_VEL
LIN {X 0,Y 565.553,Z 485.158,A -85,B 0,C 180,E1 26416.966,E2 26416.966} C_VEL
LIN {X 0,Y 565.057,Z 507.193,A -85,B 0,C 180,E1 26416.249,E2 26416.249} C_VEL
LIN {X 0,Y 564.554,Z 528.43,A -85,B 0,C 180,E1 26415.356,E2 26415.356} C_VEL
LIN {X 0,Y 563.915,Z 548.354,A -85,B 0,C 180,E1 26414.314,E2 26414.314} C_VEL
LIN {X 0,Y 563.324,Z 567.675,A -85,B 0,C 180,E1 26413.106,E2 26413.106} C_VEL
LIN {X 0,Y 562.666,Z 587.268,A -85,B 0,C 180,E1 26411.652,E2 26411.652} C_VEL
LIN {X 0,Y 562.084,Z 604.542,A -85,B 0,C 180,E1 26410.153,E2 26410.153} C_VEL
LIN {X 0,Y 561.544,Z 621.717,A -85,B 0,C 180,E1 26408.42,E2 26408.42} C_VEL
LIN {X 0,Y 561.076,Z 637.188,A -85,B 0,C 180,E1 26406.599,E2 26406.599} C_VEL
LIN {X 0,Y 560.686,Z 652.1,A -85,B 0,C 180,E1 26404.547,E2 26404.547} C_VEL
LIN {X 0,Y 560.409,Z 664.228,A -85,B 0,C 180,E1 26402.603,E2 26402.603} C_VEL
LIN {X 0,Y 560.189,Z 675.534,A -85,B 0,C 180,E1 26400.447,E2 26400.447} C_VEL
LIN {X 0,Y 560.053,Z 684.665,A -85,B 0,C 180,E1 26398.339,E2 26398.339} C_VEL
LIN {X 0,Y 559.975,Z 692.581,A -85,B 0,C 180,E1 26396.086,E2 26396.086} C_VEL
LIN {X 0,Y 559.938,Z 698.187,A -85,B 0,C 180,E1 26394.025,E2 26394.025} C_VEL
LIN {X 0,Y 559.915,Z 702.617,A -85,B 0,C 180,E1 26391.784,E2 26391.784} C_VEL
LIN {X 0,Y 559.9,Z 705.316,A -85,B 0,C 180,E1 26389.617,E2 26389.617} C_VEL
LIN {X 0,Y 559.901,Z 706.398,A -85,B 0,C 180,E1 26387.458,E2 26387.458} C_VEL
LIN {X 0,Y 559.914,Z 705.891,A -85,B 0,C 180,E1 26385.113,E2 26385.113} C_VEL
LIN {X 0,Y 559.912,Z 703.908,A -85,B 0,C 180,E1 26383.003,E2 26383.003} C_VEL
LIN {X 0,Y 559.915,Z 700.214,A -85,B 0,C 180,E1 26380.807,E2 26380.807} C_VEL
LIN {X 0,Y 559.941,Z 694.636,A -85,B 0,C 180,E1 26378.523,E2 26378.523} C_VEL
LIN {X 0,Y 560.01,Z 688.023,A -85,B 0,C 180,E1 26376.459,E2 26376.459} C_VEL
LIN {X 0,Y 560.12,Z 679.356,A -85,B 0,C 180,E1 26374.3,E2 26374.3} C_VEL
LIN {X 0,Y 560.299,Z 668.87,A -85,B 0,C 180,E1 26372.148,E2 26372.148} C_VEL
LIN {X 0,Y 560.559,Z 656.991,A -85,B 0,C 180,E1 26370.102,E2 26370.102} C_VEL
LIN {X 0,Y 560.897,Z 643.662,A -85,B 0,C 180,E1 26368.161,E2 26368.161} C_VEL
LIN {X 0,Y 561.348,Z 628.202,A -85,B 0,C 180,E1 26366.221,E2 26366.221} C_VEL
LIN {X 0,Y 561.866,Z 611.55,A -85,B 0,C 180,E1 26364.435,E2 26364.435} C_VEL
LIN {X 0,Y 562.443,Z 593.837,A -85,B 0,C 180,E1 26362.8,E2 26362.8} C_VEL
LIN {X 0,Y 563.029,Z 576.396,A -85,B 0,C 180,E1 26361.421,E2 26361.421} C_VEL
LIN {X 0,Y 563.648,Z 557.522,A -85,B 0,C 180,E1 26360.144,E2 26360.144} C_VEL
LIN {X 0,Y 564.261,Z 536.734,A -85,B 0,C 180,E1 26358.967,E2 26358.967} C_VEL
LIN {X 0,Y 564.834,Z 516.961,A -85,B 0,C 180,E1 26358.047,E2 26358.047} C_VEL
LIN {X 0,Y 565.359,Z 494.54,A -85,B 0,C 180,E1 26357.222,E2 26357.222} C_VEL
LIN {X 0,Y 565.793,Z 472.103,A -85,B 0,C 180,E1 26356.615,E2 26356.615} C_VEL
LIN {X 0,Y 566.071,Z 450.035,A -85,B 0,C 180,E1 26356.21,E2 26356.21} C_VEL
LIN {X 0,Y 567.21,Z 244.597,A -85,B 0,C 180,E1 26353.267,E2 26353.267} C_VEL
LIN {X 0,Y 567.457,Z 184.913,A -85,B 0,C 180,E1 26352.39,E2 26352.39} C_VEL
LIN {X 0,Y 561.678,Z 175.639,A -85,B 0,C 180,E1 26351.841,E2 26351.841} C_VEL
LIN {X 0,Y 560.277,Z 172.226,A -85,B 0,C 180,E1 26351.688,E2 26351.688} C_VEL
LIN {X 0,Y 560.245,Z 171.951,A -85,B 0,C 180,E1 26351.586,E2 26351.586} C_VEL
LIN {X 0,Y 560.25,Z 171.946,A -85,B 0,C 180,E1 26348.32,E2 26348.32} C_VEL
LIN {X 0,Y 560.277,Z 171.943,A -85,B 0,C 180,E1 26345.036,E2 26345.036} C_VEL
LIN {X 0,Y 560.255,Z 171.944,A -85,B 0,C 180,E1 26341.623,E2 26341.623} C_VEL
LIN {X 0,Y 560.273,Z 171.944,A -85,B 0,C 180,E1 26338.349,E2 26338.349} C_VEL
LIN {X 0,Y 560.238,Z 171.947,A -85,B 0,C 180,E1 26335.173,E2 26335.173} C_VEL
LIN {X 0,Y 560.221,Z 171.944,A -85,B 0,C 180,E1 26331.914,E2 26331.914} C_VEL
LIN {X 0,Y 560.273,Z 171.938,A -85,B 0,C 180,E1 26328.677,E2 26328.677} C_VEL
LIN {X 0,Y 560.274,Z 171.941,A -85,B 0,C 180,E1 26325.322,E2 26325.322} C_VEL
LIN {X 0,Y 560.281,Z 171.947,A -85,B 0,C 180,E1 26322.007,E2 26322.007} C_VEL
LIN {X 0,Y 560.285,Z 171.943,A -85,B 0,C 180,E1 26318.59,E2 26318.59} C_VEL
LIN {X 0,Y 560.223,Z 171.946,A -85,B 0,C 180,E1 26315.35,E2 26315.35} C_VEL
LIN {X 0,Y 560.221,Z 171.943,A -85,B 0,C 180,E1 26312.011,E2 26312.011} C_VEL
LIN {X 0,Y 560.283,Z 171.942,A -85,B 0,C 180,E1 26308.806,E2 26308.806} C_VEL
LIN {X 0,Y 560.278,Z 171.948,A -85,B 0,C 180,E1 26305.445,E2 26305.445} C_VEL
LIN {X 0,Y 560.274,Z 171.939,A -85,B 0,C 180,E1 26302.12,E2 26302.12} C_VEL
LIN {X 0,Y 560.263,Z 171.941,A -85,B 0,C 180,E1 26298.846,E2 26298.846} C_VEL
LIN {X 0,Y 560.224,Z 171.948,A -85,B 0,C 180,E1 26295.529,E2 26295.529} C_VEL
LIN {X 0,Y 560.256,Z 171.948,A -85,B 0,C 180,E1 26292.366,E2 26292.366} C_VEL
LIN {X 0,Y 560.261,Z 171.946,A -85,B 0,C 180,E1 26289.139,E2 26289.139} C_VEL
LIN {X 0,Y 560.253,Z 171.945,A -85,B 0,C 180,E1 26285.839,E2 26285.839} C_VEL
LIN {X 0,Y 560.279,Z 171.941,A -85,B 0,C 180,E1 26282.455,E2 26282.455} C_VEL
LIN {X 0,Y 560.25,Z 171.944,A -85,B 0,C 180,E1 26279.182,E2 26279.182} C_VEL
LIN {X 0,Y 560.257,Z 171.945,A -85,B 0,C 180,E1 26275.907,E2 26275.907} C_VEL
LIN {X 0,Y 560.248,Z 171.949,A -85,B 0,C 180,E1 26272.721,E2 26272.721} C_VEL
LIN {X 0,Y 560.226,Z 171.948,A -85,B 0,C 180,E1 26269.512,E2 26269.512} C_VEL
LIN {X 0,Y 560.263,Z 171.943,A -85,B 0,C 180,E1 26266.165,E2 26266.165} C_VEL
LIN {X 0,Y 560.272,Z 171.944,A -85,B 0,C 180,E1 26262.875,E2 26262.875} C_VEL
LIN {X 0,Y 560.274,Z 171.945,A -85,B 0,C 180,E1 26259.527,E2 26259.527} C_VEL
LIN {X 0,Y 560.286,Z 171.944,A -85,B 0,C 180,E1 26256.215,E2 26256.215} C_VEL
LIN {X 0,Y 560.217,Z 171.946,A -85,B 0,C 180,E1 26253.043,E2 26253.043} C_VEL
LIN {X 0,Y 560.226,Z 171.95,A -85,B 0,C 180,E1 26249.664,E2 26249.664} C_VEL
LIN {X 0,Y 560.281,Z 171.943,A -85,B 0,C 180,E1 26246.449,E2 26246.449} C_VEL
LIN {X 0,Y 560.261,Z 171.998,A -85,B 0,C 180,E1 26245.357,E2 26245.357} C_VEL
LIN {X 0,Y 561.351,Z 175.057,A -85,B 0,C 180,E1 26245.003,E2 26245.003} C_VEL
LIN {X 0,Y 564.345,Z 181.153,A -85,B 0,C 180,E1 26244.221,E2 26244.221} C_VEL
LIN {X 0,Y 568.89,Z 190.89,A -85,B 0,C 180,E1 26243.021,E2 26243.021} C_VEL
LIN {X 0,Y 567.872,Z 231.473,A -85,B 0,C 180,E1 26239.988,E2 26239.988} C_VEL
LIN {X 0,Y 567.376,Z 270.284,A -85,B 0,C 180,E1 26237.139,E2 26237.139} C_VEL
LIN {X 0,Y 568.909,Z 281.952,A -85,B 0,C 180,E1 26236.176,E2 26236.176} C_VEL
LIN {X 0,Y 572.074,Z 292.035,A -85,B 0,C 180,E1 26235.223,E2 26235.223} C_VEL
LIN {X 0,Y 575.901,Z 298.827,A -85,B 0,C 180,E1 26234.475,E2 26234.475} C_VEL
LIN {X 0,Y 581.118,Z 304.484,A -85,B 0,C 180,E1 26233.727,E2 26233.727} C_VEL
LIN {X 0,Y 584.794,Z 307.078,A -85,B 0,C 180,E1 26233.251,E2 26233.251} C_VEL
LIN {X 0,Y 587.928,Z 308.328,A -85,B 0,C 180,E1 26232.72,E2 26232.72} C_VEL
LIN {X 0,Y 590.361,Z 308.195,A -85,B 0,C 180,E1 26232.114,E2 26232.114} C_VEL
LIN {X 0,Y 591.626,Z 306.602,A -85,B 0,C 180,E1 26231.49,E2 26231.49} C_VEL
LIN {X 0,Y 591.536,Z 303.839,A -85,B 0,C 180,E1 26230.918,E2 26230.918} C_VEL
LIN {X 0,Y 590.14,Z 299.93,A -85,B 0,C 180,E1 26230.411,E2 26230.411} C_VEL
LIN {X 0,Y 587.499,Z 295.112,A -85,B 0,C 180,E1 26230.008,E2 26230.008} C_VEL
LIN {X 0,Y 583.341,Z 286.374,A -85,B 0,C 180,E1 26229.519,E2 26229.519} C_VEL
LIN {X 0,Y 580.134,Z 276.16,A -85,B 0,C 180,E1 26229.133,E2 26229.133} C_VEL
LIN {X 0,Y 577.991,Z 264.63,A -85,B 0,C 180,E1 26228.871,E2 26228.871} C_VEL
LIN {X 0,Y 576.884,Z 251.171,A -85,B 0,C 180,E1 26228.735,E2 26228.735} C_VEL
LIN {X 0,Y 576.718,Z 192.282,A -85,B 0,C 180,E1 26228.714,E2 26228.714} C_VEL
LIN {X 0,Y 574.07,Z 189.085,A -85,B 0,C 180,E1 26228.383,E2 26228.383} C_VEL
LIN {X 0,Y 573.372,Z 188.698,A -85,B 0,C 180,E1 26228.295,E2 26228.295} C_VEL
LIN {X 0,Y 569.291,Z 193.529,A -85,B 0,C 180,E1 26227.772,E2 26227.772} C_VEL
LIN {X 0,Y 567.611,Z 194.254,A -85,B 0,C 180,E1 26227.552,E2 26227.552} C_VEL
LIN {X 0,Y 566.685,Z 194.056,A -85,B 0,C 180,E1 26227.417,E2 26227.417} C_VEL
LIN {X 0,Y 566.03,Z 227.14,A -85,B 0,C 180,E1 26225.085,E2 26225.085} C_VEL
LIN {X 0,Y 567.762,Z 237.141,A -85,B 0,C 180,E1 26224.811,E2 26224.811} C_VEL
LIN {X 0,Y 566.424,Z 455.966,A -85,B 0,C 180,E1 26221.654,E2 26221.654} C_VEL
LIN {X 0,Y 565.95,Z 532.934,A -85,B 0,C 180,E1 26220.533,E2 26220.533} C_VEL
LIN {X 0,Y 565.562,Z 555.319,A -85,B 0,C 180,E1 26220.009,E2 26220.009} C_VEL
LIN {X 0,Y 565.057,Z 577.939,A -85,B 0,C 180,E1 26219.267,E2 26219.267} C_VEL
LIN {X 0,Y 564.544,Z 598.574,A -85,B 0,C 180,E1 26218.394,E2 26218.394} C_VEL
LIN {X 0,Y 563.915,Z 618.768,A -85,B 0,C 180,E1 26217.337,E2 26217.337} C_VEL
LIN {X 0,Y 563.285,Z 638.676,A -85,B 0,C 180,E1 26216.081,E2 26216.081} C_VEL
LIN {X 0,Y 562.667,Z 657.477,A -85,B 0,C 180,E1 26214.683,E2 26214.683} C_VEL
LIN {X 0,Y 562.043,Z 676.273,A -85,B 0,C 180,E1 26213.04,E2 26213.04} C_VEL
LIN {X 0,Y 561.474,Z 693.733,A -85,B 0,C 180,E1 26211.247,E2 26211.247} C_VEL
LIN {X 0,Y 561.017,Z 709.434,A -85,B 0,C 180,E1 26209.359,E2 26209.359} C_VEL
LIN {X 0,Y 560.656,Z 723.223,A -85,B 0,C 180,E1 26207.427,E2 26207.427} C_VEL
LIN {X 0,Y 560.379,Z 735.523,A -85,B 0,C 180,E1 26205.418,E2 26205.418} C_VEL
LIN {X 0,Y 560.18,Z 746.405,A -85,B 0,C 180,E1 26203.312,E2 26203.312} C_VEL
LIN {X 0,Y 560.045,Z 755.309,A -85,B 0,C 180,E1 26201.221,E2 26201.221} C_VEL
LIN {X 0,Y 559.965,Z 763.173,A -85,B 0,C 180,E1 26198.937,E2 26198.937} C_VEL
LIN {X 0,Y 559.935,Z 768.923,A -85,B 0,C 180,E1 26196.768,E2 26196.768} C_VEL
LIN {X 0,Y 559.918,Z 772.954,A -85,B 0,C 180,E1 26194.609,E2 26194.609} C_VEL
LIN {X 0,Y 559.91,Z 775.559,A -85,B 0,C 180,E1 26192.354,E2 26192.354} C_VEL
LIN {X 0,Y 559.911,Z 776.489,A -85,B 0,C 180,E1 26190.102,E2 26190.102} C_VEL
LIN {X 0,Y 559.912,Z 775.693,A -85,B 0,C 180,E1 26187.851,E2 26187.851} C_VEL
LIN {X 0,Y 559.914,Z 773.271,A -85,B 0,C 180,E1 26185.596,E2 26185.596} C_VEL
LIN {X 0,Y 559.921,Z 769.378,A -85,B 0,C 180,E1 26183.437,E2 26183.437} C_VEL
LIN {X 0,Y 559.95,Z 763.78,A -85,B 0,C 180,E1 26181.27,E2 26181.27} C_VEL
LIN {X 0,Y 560.024,Z 756.531,A -85,B 0,C 180,E1 26179.091,E2 26179.091} C_VEL
LIN {X 0,Y 560.159,Z 747.379,A -85,B 0,C 180,E1 26176.898,E2 26176.898} C_VEL
LIN {X 0,Y 560.347,Z 736.679,A -85,B 0,C 180,E1 26174.793,E2 26174.793} C_VEL
LIN {X 0,Y 560.637,Z 723.881,A -85,B 0,C 180,E1 26172.672,E2 26172.672} C_VEL
LIN {X 0,Y 560.996,Z 710.279,A -85,B 0,C 180,E1 26170.748,E2 26170.748} C_VEL
LIN {X 0,Y 561.461,Z 694.221,A -85,B 0,C 180,E1 26168.807,E2 26168.807} C_VEL
LIN {X 0,Y 562.023,Z 676.828,A -85,B 0,C 180,E1 26167.014,E2 26167.014} C_VEL
LIN {X 0,Y 562.625,Z 658.817,A -85,B 0,C 180,E1 26165.427,E2 26165.427} C_VEL
LIN {X 0,Y 563.244,Z 639.765,A -85,B 0,C 180,E1 26163.993,E2 26163.993} C_VEL
LIN {X 0,Y 563.892,Z 619.755,A -85,B 0,C 180,E1 26162.719,E2 26162.719} C_VEL
LIN {X 0,Y 564.5,Z 599.709,A -85,B 0,C 180,E1 26161.661,E2 26161.661} C_VEL
LIN {X 0,Y 565.033,Z 578.77,A -85,B 0,C 180,E1 26160.764,E2 26160.764} C_VEL
LIN {X 0,Y 565.546,Z 556.44,A -85,B 0,C 180,E1 26160.023,E2 26160.023} C_VEL
LIN {X 0,Y 565.924,Z 534.15,A -85,B 0,C 180,E1 26159.491,E2 26159.491} C_VEL
LIN {X 0,Y 566.231,Z 490.039,A -85,B 0,C 180,E1 26158.83,E2 26158.83} C_VEL
LIN {X 0,Y 567.542,Z 270.808,A -85,B 0,C 180,E1 26155.68,E2 26155.68} C_VEL
LIN {X 0,Y 567.591,Z 230.761,A -85,B 0,C 180,E1 26155.08,E2 26155.08} C_VEL
LIN {X 0,Y 566.847,Z 224.044,A -85,B 0,C 180,E1 26154.898,E2 26154.898} C_VEL
LIN {X 0,Y 567.453,Z 187.335,A -85,B 0,C 180,E1 26153.079,E2 26153.079} C_VEL
LIN {X 0,Y 565.6,Z 183.409,A -85,B 0,C 180,E1 26152.713,E2 26152.713} C_VEL
LIN {X 0,Y 567.614,Z 183.633,A -85,B 0,C 180,E1 26152.448,E2 26152.448} C_VEL
LIN {X 0,Y 568.834,Z 183.271,A -85,B 0,C 180,E1 26152.288,E2 26152.288} C_VEL
LIN {X 0,Y 570.443,Z 184.778,A -85,B 0,C 180,E1 26152.079,E2 26152.079} C_VEL
LIN {X 0,Y 574.072,Z 189.073,A -85,B 0,C 180,E1 26151.617,E2 26151.617} C_VEL
LIN {X 0,Y 581.282,Z 197.483,A -85,B 0,C 180,E1 26150.728,E2 26150.728} C_VEL
LIN {X 0,Y 589.596,Z 206.471,A -85,B 0,C 180,E1 26149.75,E2 26149.75} C_VEL
LIN {X 0,Y 592.95,Z 209.312,A -85,B 0,C 180,E1 26149.263,E2 26149.263} C_VEL
LIN {X 0,Y 594.973,Z 211.203,A -85,B 0,C 180,E1 26148.693,E2 26148.693} C_VEL
LIN {X 0,Y 595.613,Z 212.159,A -85,B 0,C 180,E1 26148.044,E2 26148.044} C_VEL
LIN {X 0,Y 594.548,Z 213.078,A -85,B 0,C 180,E1 26147.441,E2 26147.441} C_VEL
LIN {X 0,Y 592.148,Z 212.827,A -85,B 0,C 180,E1 26146.839,E2 26146.839} C_VEL
LIN {X 0,Y 588.922,Z 211.334,A -85,B 0,C 180,E1 26146.323,E2 26146.323} C_VEL
LIN {X 0,Y 583.742,Z 207.462,A -85,B 0,C 180,E1 26145.722,E2 26145.722} C_VEL
LIN {X 0,Y 577.102,Z 202.352,A -85,B 0,C 180,E1 26144.981,E2 26144.981} C_VEL
LIN {X 0,Y 572.392,Z 196.466,A -85,B 0,C 180,E1 26144.324,E2 26144.324} C_VEL
LIN {X 0,Y 561.929,Z 175.946,A -85,B 0,C 180,E1 26142.402,E2 26142.402} C_VEL
LIN {X 0,Y 560.483,Z 173.097,A -85,B 0,C 180,E1 26142.125,E2 26142.125} C_VEL
LIN {X 0,Y 560.259,Z 171.946,A -85,B 0,C 180,E1 26142.008,E2 26142.008} C_VEL
LIN {X 0,Y 560.243,Z 171.943,A -85,B 0,C 180,E1 26138.655,E2 26138.655} C_VEL
LIN {X 0,Y 560.28,Z 171.941,A -85,B 0,C 180,E1 26135.358,E2 26135.358} C_VEL
LIN {X 0,Y 560.242,Z 171.947,A -85,B 0,C 180,E1 26132.129,E2 26132.129} C_VEL
LIN {X 0,Y 560.294,Z 172.018,A -85,B 0,C 180,E1 26131.524,E2 26131.524} C_VEL
LIN {X 0,Y 561.23,Z 177.579,A -85,B 0,C 180,E1 26131.107,E2 26131.107} C_VEL
LIN {X 0,Y 562.068,Z 211.516,A -85,B 0,C 180,E1 26128.589,E2 26128.589} C_VEL
LIN {X 0,Y 562.344,Z 242.353,A -85,B 0,C 180,E1 26126.116,E2 26126.116} C_VEL
LIN {X 0,Y 562.269,Z 271.353,A -85,B 0,C 180,E1 26123.679,E2 26123.679} C_VEL
LIN {X 0,Y 561.847,Z 299.179,A -85,B 0,C 180,E1 26121.258,E2 26121.258} C_VEL
LIN {X 0,Y 561.666,Z 313.467,A -85,B 0,C 180,E1 26120.028,E2 26120.028} C_VEL
LIN {X 0,Y 562.479,Z 320.667,A -85,B 0,C 180,E1 26119.907,E2 26119.907} C_VEL
LIN {X 0,Y 561.938,Z 481.52,A -85,B 0,C 180,E1 26117.77,E2 26117.77} C_VEL
LIN {X 0,Y 561.808,Z 498.664,A -85,B 0,C 180,E1 26117.367,E2 26117.367} C_VEL
LIN {X 0,Y 561.594,Z 515.172,A -85,B 0,C 180,E1 26116.79,E2 26116.79} C_VEL
LIN {X 0,Y 561.326,Z 531.318,A -85,B 0,C 180,E1 26116.027,E2 26116.027} C_VEL
LIN {X 0,Y 561.053,Z 546.167,A -85,B 0,C 180,E1 26115.134,E2 26115.134} C_VEL
LIN {X 0,Y 560.77,Z 561.444,A -85,B 0,C 180,E1 26113.981,E2 26113.981} C_VEL
LIN {X 0,Y 560.499,Z 575.738,A -85,B 0,C 180,E1 26112.635,E2 26112.635} C_VEL
LIN {X 0,Y 560.283,Z 587.926,A -85,B 0,C 180,E1 26111.216,E2 26111.216} C_VEL
LIN {X 0,Y 560.132,Z 598.072,A -85,B 0,C 180,E1 26109.763,E2 26109.763} C_VEL
LIN {X 0,Y 560.026,Z 606.841,A -85,B 0,C 180,E1 26108.211,E2 26108.211} C_VEL
LIN {X 0,Y 559.959,Z 614.558,A -85,B 0,C 180,E1 26106.459,E2 26106.459} C_VEL
LIN {X 0,Y 559.93,Z 620.197,A -85,B 0,C 180,E1 26104.711,E2 26104.711} C_VEL
LIN {X 0,Y 559.915,Z 623.977,A -85,B 0,C 180,E1 26102.968,E2 26102.968} C_VEL
LIN {X 0,Y 559.915,Z 626.039,A -85,B 0,C 180,E1 26101.228,E2 26101.228} C_VEL
LIN {X 0,Y 559.917,Z 626.394,A -85,B 0,C 180,E1 26099.386,E2 26099.386} C_VEL
LIN {X 0,Y 559.911,Z 625.018,A -85,B 0,C 180,E1 26097.646,E2 26097.646} C_VEL
LIN {X 0,Y 559.918,Z 621.949,A -85,B 0,C 180,E1 26095.904,E2 26095.904} C_VEL
LIN {X 0,Y 559.942,Z 616.716,A -85,B 0,C 180,E1 26094.055,E2 26094.055} C_VEL
LIN {X 0,Y 560.001,Z 609.744,A -85,B 0,C 180,E1 26092.304,E2 26092.304} C_VEL
LIN {X 0,Y 560.086,Z 601.749,A -85,B 0,C 180,E1 26090.754,E2 26090.754} C_VEL
LIN {X 0,Y 560.224,Z 591.699,A -85,B 0,C 180,E1 26089.199,E2 26089.199} C_VEL
LIN {X 0,Y 560.421,Z 580.025,A -85,B 0,C 180,E1 26087.742,E2 26087.742} C_VEL
LIN {X 0,Y 560.645,Z 567.743,A -85,B 0,C 180,E1 26086.489,E2 26086.489} C_VEL
LIN {X 0,Y 560.911,Z 554.021,A -85,B 0,C 180,E1 26085.337,E2 26085.337} C_VEL
LIN {X 0,Y 561.199,Z 538.48,A -85,B 0,C 180,E1 26084.287,E2 26084.287} C_VEL
LIN {X 0,Y 561.46,Z 522.579,A -85,B 0,C 180,E1 26083.445,E2 26083.445} C_VEL
LIN {X 0,Y 561.7,Z 507.024,A -85,B 0,C 180,E1 26082.813,E2 26082.813} C_VEL
LIN {X 0,Y 561.899,Z 490.227,A -85,B 0,C 180,E1 26082.322,E2 26082.322} C_VEL
LIN {X 0,Y 561.296,Z 483.791,A -85,B 0,C 180,E1 26082.158,E2 26082.158} C_VEL
LIN {X 0,Y 556.857,Z 469.234,A -85,B 0,C 180,E1 26081.779,E2 26081.779} C_VEL
LIN {X 0,Y 554.764,Z 460.737,A -85,B 0,C 180,E1 26081.603,E2 26081.603} C_VEL
LIN {X 0,Y 554.447,Z 456.358,A -85,B 0,C 180,E1 26081.537,E2 26081.537} C_VEL
LIN {X 0,Y 554.74,Z 318.575,A -85,B 0,C 180,E1 26079.706,E2 26079.706} C_VEL
LIN {X 0,Y 553.983,Z 313.922,A -85,B 0,C 180,E1 26079.614,E2 26079.614} C_VEL
LIN {X 0,Y 554.576,Z 279.08,A -85,B 0,C 180,E1 26076.462,E2 26076.462} C_VEL
LIN {X 0,Y 555.017,Z 243.083,A -85,B 0,C 180,E1 26073.232,E2 26073.232} C_VEL
LIN {X 0,Y 555.312,Z 209.757,A -85,B 0,C 180,E1 26070.255,E2 26070.255} C_VEL
LIN {X 0,Y 555.348,Z 183.324,A -85,B 0,C 180,E1 26067.918,E2 26067.918} C_VEL
LIN {X 0,Y 552.334,Z 172.938,A -85,B 0,C 180,E1 26066.797,E2 26066.797} C_VEL
LIN {X 0,Y 552.332,Z 172.934,A -85,B 0,C 180,E1 26063.446,E2 26063.446} C_VEL
LIN {X 0,Y 552.355,Z 173.054,A -85,B 0,C 180,E1 26062.792,E2 26062.792} C_VEL
LIN {X 0,Y 553.658,Z 176.446,A -85,B 0,C 180,E1 26062.642,E2 26062.642} C_VEL
LIN {X 0,Y 555.399,Z 179.169,A -85,B 0,C 180,E1 26062.471,E2 26062.471} C_VEL
LIN {X 0,Y 561.037,Z 188.688,A -85,B 0,C 180,E1 26061.915,E2 26061.915} C_VEL
LIN {X 0,Y 559.436,Z 411.946,A -85,B 0,C 180,E1 26058.667,E2 26058.667} C_VEL
LIN {X 0,Y 559.046,Z 463.901,A -85,B 0,C 180,E1 26057.888,E2 26057.888} C_VEL
LIN {X 0,Y 558.583,Z 485.472,A -85,B 0,C 180,E1 26057.371,E2 26057.371} C_VEL
LIN {X 0,Y 558.01,Z 507.522,A -85,B 0,C 180,E1 26056.643,E2 26056.643} C_VEL
LIN {X 0,Y 557.412,Z 528.48,A -85,B 0,C 180,E1 26055.751,E2 26055.751} C_VEL
LIN {X 0,Y 556.649,Z 549.059,A -85,B 0,C 180,E1 26054.659,E2 26054.659} C_VEL
LIN {X 0,Y 555.93,Z 568.856,A -85,B 0,C 180,E1 26053.397,E2 26053.397} C_VEL
LIN {X 0,Y 555.155,Z 588.221,A -85,B 0,C 180,E1 26051.928,E2 26051.928} C_VEL
LIN {X 0,Y 554.491,Z 605.319,A -85,B 0,C 180,E1 26050.417,E2 26050.417} C_VEL
LIN {X 0,Y 553.846,Z 622.4,A -85,B 0,C 180,E1 26048.656,E2 26048.656} C_VEL
LIN {X 0,Y 553.297,Z 637.723,A -85,B 0,C 180,E1 26046.817,E2 26046.817} C_VEL
LIN {X 0,Y 552.842,Z 652.104,A -85,B 0,C 180,E1 26044.805,E2 26044.805} C_VEL
LIN {X 0,Y 552.505,Z 663.94,A -85,B 0,C 180,E1 26042.882,E2 26042.882} C_VEL
LIN {X 0,Y 552.246,Z 675.358,A -85,B 0,C 180,E1 26040.682,E2 26040.682} C_VEL
LIN {X 0,Y 552.08,Z 684.485,A -85,B 0,C 180,E1 26038.553,E2 26038.553} C_VEL
LIN {X 0,Y 551.99,Z 692.403,A -85,B 0,C 180,E1 26036.281,E2 26036.281} C_VEL
LIN {X 0,Y 551.943,Z 698.092,A -85,B 0,C 180,E1 26034.168,E2 26034.168} C_VEL
LIN {X 0,Y 551.917,Z 702.531,A -85,B 0,C 180,E1 26031.913,E2 26031.913} C_VEL
LIN {X 0,Y 551.902,Z 705.358,A -85,B 0,C 180,E1 26029.598,E2 26029.598} C_VEL
LIN {X 0,Y 551.901,Z 706.39,A -85,B 0,C 180,E1 26027.502,E2 26027.502} C_VEL
LIN {X 0,Y 551.913,Z 705.916,A -85,B 0,C 180,E1 26025.122,E2 26025.122} C_VEL
LIN {X 0,Y 551.911,Z 703.877,A -85,B 0,C 180,E1 26022.925,E2 26022.925} C_VEL
LIN {X 0,Y 551.916,Z 700.288,A -85,B 0,C 180,E1 26020.754,E2 26020.754} C_VEL
LIN {X 0,Y 551.949,Z 694.741,A -85,B 0,C 180,E1 26018.438,E2 26018.438} C_VEL
LIN {X 0,Y 552.029,Z 688.152,A -85,B 0,C 180,E1 26016.344,E2 26016.344} C_VEL
LIN {X 0,Y 552.163,Z 679.53,A -85,B 0,C 180,E1 26014.154,E2 26014.154} C_VEL
LIN {X 0,Y 552.379,Z 669.085,A -85,B 0,C 180,E1 26011.971,E2 26011.971} C_VEL
LIN {X 0,Y 552.701,Z 656.585,A -85,B 0,C 180,E1 26009.793,E2 26009.793} C_VEL
LIN {X 0,Y 553.086,Z 643.961,A -85,B 0,C 180,E1 26007.928,E2 26007.928} C_VEL
LIN {X 0,Y 553.622,Z 628.564,A -85,B 0,C 180,E1 26005.961,E2 26005.961} C_VEL
LIN {X 0,Y 554.236,Z 611.969,A -85,B 0,C 180,E1 26004.15,E2 26004.15} C_VEL
LIN {X 0,Y 554.926,Z 594.331,A -85,B 0,C 180,E1 26002.494,E2 26002.494} C_VEL
LIN {X 0,Y 555.627,Z 576.245,A -85,B 0,C 180,E1 26001.045,E2 26001.045} C_VEL
LIN {X 0,Y 556.372,Z 557.34,A -85,B 0,C 180,E1 25999.752,E2 25999.752} C_VEL
LIN {X 0,Y 557.056,Z 537.483,A -85,B 0,C 180,E1 25998.613,E2 25998.613} C_VEL
LIN {X 0,Y 557.685,Z 518.703,A -85,B 0,C 180,E1 25997.721,E2 25997.721} C_VEL
LIN {X 0,Y 558.304,Z 496.849,A -85,B 0,C 180,E1 25996.887,E2 25996.887} C_VEL
LIN {X 0,Y 558.844,Z 474.86,A -85,B 0,C 180,E1 25996.26,E2 25996.26} C_VEL
LIN {X 0,Y 559.147,Z 453.171,A -85,B 0,C 180,E1 25995.839,E2 25995.839} C_VEL
LIN {X 0,Y 560.525,Z 248.274,A -85,B 0,C 180,E1 25992.866,E2 25992.866} C_VEL
LIN {X 0,Y 560.853,Z 188.138,A -85,B 0,C 180,E1 25991.973,E2 25991.973} C_VEL
LIN {X 0,Y 553.938,Z 176.834,A -85,B 0,C 180,E1 25991.295,E2 25991.295} C_VEL
LIN {X 0,Y 552.425,Z 173.453,A -85,B 0,C 180,E1 25991.129,E2 25991.129} C_VEL
LIN {X 0,Y 552.344,Z 172.936,A -85,B 0,C 180,E1 25991.093,E2 25991.093} C_VEL
LIN {X 0,Y 552.334,Z 172.936,A -85,B 0,C 180,E1 25987.675,E2 25987.675} C_VEL
LIN {X 0,Y 552.33,Z 172.935,A -85,B 0,C 180,E1 25984.358,E2 25984.358} C_VEL
LIN {X 0,Y 552.334,Z 172.929,A -85,B 0,C 180,E1 25980.978,E2 25980.978} C_VEL
LIN {X 0,Y 552.293,Z 172.935,A -85,B 0,C 180,E1 25977.72,E2 25977.72} C_VEL
LIN {X 0,Y 552.307,Z 172.938,A -85,B 0,C 180,E1 25974.471,E2 25974.471} C_VEL
LIN {X 0,Y 552.324,Z 172.933,A -85,B 0,C 180,E1 25971.218,E2 25971.218} C_VEL
LIN {X 0,Y 552.311,Z 172.93,A -85,B 0,C 180,E1 25967.922,E2 25967.922} C_VEL
LIN {X 0,Y 552.332,Z 172.926,A -85,B 0,C 180,E1 25964.501,E2 25964.501} C_VEL
LIN {X 0,Y 552.317,Z 172.929,A -85,B 0,C 180,E1 25961.22,E2 25961.22} C_VEL
LIN {X 0,Y 552.305,Z 172.935,A -85,B 0,C 180,E1 25957.858,E2 25957.858} C_VEL
LIN {X 0,Y 552.333,Z 172.938,A -85,B 0,C 180,E1 25954.547,E2 25954.547} C_VEL
LIN {X 0,Y 552.301,Z 172.932,A -85,B 0,C 180,E1 25951.297,E2 25951.297} C_VEL
LIN {X 0,Y 552.306,Z 172.932,A -85,B 0,C 180,E1 25947.962,E2 25947.962} C_VEL
LIN {X 0,Y 552.339,Z 172.93,A -85,B 0,C 180,E1 25944.605,E2 25944.605} C_VEL
LIN {X 0,Y 552.321,Z 172.935,A -85,B 0,C 180,E1 25941.338,E2 25941.338} C_VEL
LIN {X 0,Y 552.334,Z 172.931,A -85,B 0,C 180,E1 25938.033,E2 25938.033} C_VEL
LIN {X 0,Y 552.331,Z 172.936,A -85,B 0,C 180,E1 25934.681,E2 25934.681} C_VEL
LIN {X 0,Y 552.283,Z 172.937,A -85,B 0,C 180,E1 25931.382,E2 25931.382} C_VEL
LIN {X 0,Y 552.303,Z 172.931,A -85,B 0,C 180,E1 25928.004,E2 25928.004} C_VEL
LIN {X 0,Y 552.337,Z 172.926,A -85,B 0,C 180,E1 25924.777,E2 25924.777} C_VEL
LIN {X 0,Y 552.328,Z 172.933,A -85,B 0,C 180,E1 25921.349,E2 25921.349} C_VEL
LIN {X 0,Y 552.341,Z 172.936,A -85,B 0,C 180,E1 25918.029,E2 25918.029} C_VEL
LIN {X 0,Y 552.316,Z 172.932,A -85,B 0,C 180,E1 25914.703,E2 25914.703} C_VEL
LIN {X 0,Y 552.273,Z 172.934,A -85,B 0,C 180,E1 25911.463,E2 25911.463} C_VEL
LIN {X 0,Y 552.32,Z 172.93,A -85,B 0,C 180,E1 25908.196,E2 25908.196} C_VEL
LIN {X 0,Y 552.34,Z 172.931,A -85,B 0,C 180,E1 25904.89,E2 25904.89} C_VEL
LIN {X 0,Y 552.341,Z 172.932,A -85,B 0,C 180,E1 25901.532,E2 25901.532} C_VEL
LIN {X 0,Y 552.342,Z 172.929,A -85,B 0,C 180,E1 25898.105,E2 25898.105} C_VEL
LIN {X 0,Y 552.3,Z 172.936,A -85,B 0,C 180,E1 25894.847,E2 25894.847} C_VEL
LIN {X 0,Y 552.272,Z 172.939,A -85,B 0,C 180,E1 25891.448,E2 25891.448} C_VEL
LIN {X 0,Y 552.332,Z 172.935,A -85,B 0,C 180,E1 25888.212,E2 25888.212} C_VEL
LIN {X 0,Y 552.329,Z 172.973,A -85,B 0,C 180,E1 25886.077,E2 25886.077} C_VEL
LIN {X 0,Y 553.477,Z 176.208,A -85,B 0,C 180,E1 25885.693,E2 25885.693} C_VEL
LIN {X 0,Y 556.48,Z 182.221,A -85,B 0,C 180,E1 25884.903,E2 25884.903} C_VEL
LIN {X 0,Y 562.399,Z 195.047,A -85,B 0,C 180,E1 25883.303,E2 25883.303} C_VEL
LIN {X 0,Y 561.211,Z 235.727,A -85,B 0,C 180,E1 25880.239,E2 25880.239} C_VEL
LIN {X 0,Y 560.608,Z 273.015,A -85,B 0,C 180,E1 25877.472,E2 25877.472} C_VEL
LIN {X 0,Y 562.175,Z 285.437,A -85,B 0,C 180,E1 25876.434,E2 25876.434} C_VEL
LIN {X 0,Y 565.225,Z 295.574,A -85,B 0,C 180,E1 25875.47,E2 25875.47} C_VEL
LIN {X 0,Y 569.305,Z 303.253,A -85,B 0,C 180,E1 25874.629,E2 25874.629} C_VEL
LIN {X 0,Y 574.867,Z 309.628,A -85,B 0,C 180,E1 25873.797,E2 25873.797} C_VEL
LIN {X 0,Y 580.653,Z 313.822,A -85,B 0,C 180,E1 25873.105,E2 25873.105} C_VEL
LIN {X 0,Y 584.114,Z 315.259,A -85,B 0,C 180,E1 25872.604,E2 25872.604} C_VEL
LIN {X 0,Y 586.911,Z 315.435,A -85,B 0,C 180,E1 25872.029,E2 25872.029} C_VEL
LIN {X 0,Y 588.544,Z 314.427,A -85,B 0,C 180,E1 25871.479,E2 25871.479} C_VEL
LIN {X 0,Y 589.1,Z 312.093,A -85,B 0,C 180,E1 25870.866,E2 25870.866} C_VEL
LIN {X 0,Y 588.285,Z 308.781,A -85,B 0,C 180,E1 25870.325,E2 25870.325} C_VEL
LIN {X 0,Y 586.046,Z 304.325,A -85,B 0,C 180,E1 25869.848,E2 25869.848} C_VEL
LIN {X 0,Y 581.28,Z 295.822,A -85,B 0,C 180,E1 25869.271,E2 25869.271} C_VEL
LIN {X 0,Y 577.423,Z 286.023,A -85,B 0,C 180,E1 25868.801,E2 25868.801} C_VEL
LIN {X 0,Y 574.536,Z 274.901,A -85,B 0,C 180,E1 25868.442,E2 25868.442} C_VEL
LIN {X 0,Y 572.638,Z 262.185,A -85,B 0,C 180,E1 25868.202,E2 25868.202} C_VEL
LIN {X 0,Y 571.805,Z 247.316,A -85,B 0,C 180,E1 25868.096,E2 25868.096} C_VEL
LIN {X 0,Y 571.749,Z 200.473,A -85,B 0,C 180,E1 25868.089,E2 25868.089} C_VEL
LIN {X 0,Y 569.214,Z 202.287,A -85,B 0,C 180,E1 25867.762,E2 25867.762} C_VEL
LIN {X 0,Y 565.258,Z 210.171,A -85,B 0,C 180,E1 25867.241,E2 25867.241} C_VEL
LIN {X 0,Y 562.172,Z 214.155,A -85,B 0,C 180,E1 25866.825,E2 25866.825} C_VEL
LIN {X 0,Y 560.379,Z 215.11,A -85,B 0,C 180,E1 25866.58,E2 25866.58} C_VEL
LIN {X 0,Y 559.4,Z 214.935,A -85,B 0,C 180,E1 25866.431,E2 25866.431} C_VEL
LIN {X 0,Y 559.189,Z 227.255,A -85,B 0,C 180,E1 25865.577,E2 25865.577} C_VEL
LIN {X 0,Y 561.183,Z 238.643,A -85,B 0,C 180,E1 25865.257,E2 25865.257} C_VEL
LIN {X 0,Y 559.604,Z 457.365,A -85,B 0,C 180,E1 25862.065,E2 25862.065} C_VEL
LIN {X 0,Y 559.053,Z 532.921,A -85,B 0,C 180,E1 25860.951,E2 25860.951} C_VEL
LIN {X 0,Y 558.598,Z 555.194,A -85,B 0,C 180,E1 25860.426,E2 25860.426} C_VEL
LIN {X 0,Y 558.038,Z 577.47,A -85,B 0,C 180,E1 25859.691,E2 25859.691} C_VEL
LIN {X 0,Y 557.404,Z 598.57,A -85,B 0,C 180,E1 25858.792,E2 25858.792} C_VEL
LIN {X 0,Y 556.653,Z 619.456,A -85,B 0,C 180,E1 25857.684,E2 25857.684} C_VEL
LIN {X 0,Y 555.904,Z 639.43,A -85,B 0,C 180,E1 25856.401,E2 25856.401} C_VEL
LIN {X 0,Y 555.122,Z 659.417,A -85,B 0,C 180,E1 25854.877,E2 25854.877} C_VEL
LIN {X 0,Y 554.412,Z 677.391,A -85,B 0,C 180,E1 25853.263,E2 25853.263} C_VEL
LIN {X 0,Y 553.774,Z 694.224,A -85,B 0,C 180,E1 25851.501,E2 25851.501} C_VEL
LIN {X 0,Y 553.217,Z 710.284,A -85,B 0,C 180,E1 25849.534,E2 25849.534} C_VEL
LIN {X 0,Y 552.792,Z 723.888,A -85,B 0,C 180,E1 25847.581,E2 25847.581} C_VEL
LIN {X 0,Y 552.444,Z 736.685,A -85,B 0,C 180,E1 25845.429,E2 25845.429} C_VEL
LIN {X 0,Y 552.215,Z 747.381,A -85,B 0,C 180,E1 25843.294,E2 25843.294} C_VEL
LIN {X 0,Y 552.055,Z 756.534,A -85,B 0,C 180,E1 25841.068,E2 25841.068} C_VEL
LIN {X 0,Y 551.965,Z 763.783,A -85,B 0,C 180,E1 25838.857,E2 25838.857} C_VEL
LIN {X 0,Y 551.93,Z 769.379,A -85,B 0,C 180,E1 25836.658,E2 25836.658} C_VEL
LIN {X 0,Y 551.916,Z 773.274,A -85,B 0,C 180,E1 25834.468,E2 25834.468} C_VEL
LIN {X 0,Y 551.913,Z 775.695,A -85,B 0,C 180,E1 25832.18,E2 25832.18} C_VEL
LIN {X 0,Y 551.911,Z 776.5,A -85,B 0,C 180,E1 25830,E2 25830} C_VEL
LIN {X 0,Y 551.911,Z 775.628,A -85,B 0,C 180,E1 25827.716,E2 25827.716} C_VEL
LIN {X 0,Y 551.917,Z 773.115,A -85,B 0,C 180,E1 25825.428,E2 25825.428} C_VEL
LIN {X 0,Y 551.937,Z 769.16,A -85,B 0,C 180,E1 25823.238,E2 25823.238} C_VEL
LIN {X 0,Y 551.975,Z 763.479,A -85,B 0,C 180,E1 25821.038,E2 25821.038} C_VEL
LIN {X 0,Y 552.067,Z 755.719,A -85,B 0,C 180,E1 25818.72,E2 25818.72} C_VEL
LIN {X 0,Y 552.225,Z 746.891,A -85,B 0,C 180,E1 25816.599,E2 25816.599} C_VEL
LIN {X 0,Y 552.46,Z 736.104,A -85,B 0,C 180,E1 25814.463,E2 25814.463} C_VEL
LIN {X 0,Y 552.795,Z 723.774,A -85,B 0,C 180,E1 25812.401,E2 25812.401} C_VEL
LIN {X 0,Y 553.217,Z 710.281,A -85,B 0,C 180,E1 25810.466,E2 25810.466} C_VEL
LIN {X 0,Y 553.773,Z 694.221,A -85,B 0,C 180,E1 25808.498,E2 25808.498} C_VEL
LIN {X 0,Y 554.434,Z 676.829,A -85,B 0,C 180,E1 25806.681,E2 25806.681} C_VEL
LIN {X 0,Y 555.144,Z 658.822,A -85,B 0,C 180,E1 25805.073,E2 25805.073} C_VEL
LIN {X 0,Y 555.906,Z 639.424,A -85,B 0,C 180,E1 25803.599,E2 25803.599} C_VEL
LIN {X 0,Y 556.652,Z 619.459,A -85,B 0,C 180,E1 25802.316,E2 25802.316} C_VEL
LIN {X 0,Y 557.399,Z 598.563,A -85,B 0,C 180,E1 25801.208,E2 25801.208} C_VEL
LIN {X 0,Y 558.044,Z 577.316,A -85,B 0,C 180,E1 25800.303,E2 25800.303} C_VEL
LIN {X 0,Y 558.61,Z 554.376,A -85,B 0,C 180,E1 25799.551,E2 25799.551} C_VEL
LIN {X 0,Y 559.076,Z 531.815,A -85,B 0,C 180,E1 25799.028,E2 25799.028} C_VEL
LIN {X 0,Y 560.742,Z 297.768,A -85,B 0,C 180,E1 25795.615,E2 25795.615} C_VEL
LIN {X 0,Y 561.033,Z 232.102,A -85,B 0,C 180,E1 25794.632,E2 25794.632} C_VEL
LIN {X 0,Y 560.131,Z 224.044,A -85,B 0,C 180,E1 25794.414,E2 25794.414} C_VEL
LIN {X 0,Y 560.679,Z 203.592,A -85,B 0,C 180,E1 25793.379,E2 25793.379} C_VEL
LIN {X 0,Y 562.174,Z 203.111,A -85,B 0,C 180,E1 25793.175,E2 25793.175} C_VEL
LIN {X 0,Y 564.806,Z 199.134,A -85,B 0,C 180,E1 25792.819,E2 25792.819} C_VEL
LIN {X 0,Y 567.918,Z 191.857,A -85,B 0,C 180,E1 25792.407,E2 25792.407} C_VEL
LIN {X 0,Y 586.378,Z 212.83,A -85,B 0,C 180,E1 25790.123,E2 25790.123} C_VEL
LIN {X 0,Y 590.404,Z 216.214,A -85,B 0,C 180,E1 25789.594,E2 25789.594} C_VEL
LIN {X 0,Y 592.65,Z 218.304,A -85,B 0,C 180,E1 25789.047,E2 25789.047} C_VEL
LIN {X 0,Y 593.563,Z 219.582,A -85,B 0,C 180,E1 25788.41,E2 25788.41} C_VEL
LIN {X 0,Y 593.007,Z 220.322,A -85,B 0,C 180,E1 25787.851,E2 25787.851} C_VEL
LIN {X 0,Y 590.956,Z 220.633,A -85,B 0,C 180,E1 25787.248,E2 25787.248} C_VEL
LIN {X 0,Y 587.9,Z 219.763,A -85,B 0,C 180,E1 25786.711,E2 25786.711} C_VEL
LIN {X 0,Y 584.098,Z 217.764,A -85,B 0,C 180,E1 25786.251,E2 25786.251} C_VEL
LIN {X 0,Y 572.094,Z 208.558,A -85,B 0,C 180,E1 25784.916,E2 25784.916} C_VEL
LIN {X 0,Y 566.799,Z 201.984,A -85,B 0,C 180,E1 25784.17,E2 25784.17} C_VEL
LIN {X 0,Y 553.965,Z 176.858,A -85,B 0,C 180,E1 25781.76,E2 25781.76} C_VEL
LIN {X 0,Y 552.435,Z 173.51,A -85,B 0,C 180,E1 25781.435,E2 25781.435} C_VEL
LIN {X 0,Y 552.343,Z 172.933,A -85,B 0,C 180,E1 25781.355,E2 25781.355} C_VEL
LIN {X 0,Y 552.313,Z 172.928,A -85,B 0,C 180,E1 25778.048,E2 25778.048} C_VEL
LIN {X 0,Y 552.301,Z 172.937,A -85,B 0,C 180,E1 25774.642,E2 25774.642} C_VEL
LIN {X 0,Y 552.346,Z 173.014,A -85,B 0,C 180,E1 25771.737,E2 25771.737} C_VEL
LIN {X 0,Y 553.544,Z 179.217,A -85,B 0,C 180,E1 25771.266,E2 25771.266} C_VEL
LIN {X 0,Y 554.342,Z 210.207,A -85,B 0,C 180,E1 25768.979,E2 25768.979} C_VEL
LIN {X 0,Y 554.789,Z 243.117,A -85,B 0,C 180,E1 25766.4,E2 25766.4} C_VEL
LIN {X 0,Y 554.663,Z 279.926,A -85,B 0,C 180,E1 25763.308,E2 25763.308} C_VEL
LIN {X 0,Y 554.189,Z 315.429,A -85,B 0,C 180,E1 25760.242,E2 25760.242} C_VEL
LIN {X 0,Y 554.832,Z 321.813,A -85,B 0,C 180,E1 25760.135,E2 25760.135} C_VEL
LIN {X 0,Y 554.292,Z 481.805,A -85,B 0,C 180,E1 25758.01,E2 25758.01} C_VEL
LIN {X 0,Y 554.153,Z 498.819,A -85,B 0,C 180,E1 25757.608,E2 25757.608} C_VEL
LIN {X 0,Y 553.918,Z 514.479,A -85,B 0,C 180,E1 25757.057,E2 25757.057} C_VEL
LIN {X 0,Y 553.625,Z 530.062,A -85,B 0,C 180,E1 25756.326,E2 25756.326} C_VEL
LIN {X 0,Y 553.293,Z 545.401,A -85,B 0,C 180,E1 25755.405,E2 25755.405} C_VEL
LIN {X 0,Y 552.947,Z 560.832,A -85,B 0,C 180,E1 25754.236,E2 25754.236} C_VEL
LIN {X 0,Y 552.631,Z 574.857,A -85,B 0,C 180,E1 25752.911,E2 25752.911} C_VEL
LIN {X 0,Y 552.373,Z 587.104,A -85,B 0,C 180,E1 25751.485,E2 25751.485} C_VEL
LIN {X 0,Y 552.186,Z 597.423,A -85,B 0,C 180,E1 25750.01,E2 25750.01} C_VEL
LIN {X 0,Y 552.058,Z 606.332,A -85,B 0,C 180,E1 25748.436,E2 25748.436} C_VEL
LIN {X 0,Y 551.974,Z 614.159,A -85,B 0,C 180,E1 25746.657,E2 25746.657} C_VEL
LIN {X 0,Y 551.932,Z 619.91,A -85,B 0,C 180,E1 25744.884,E2 25744.884} C_VEL
LIN {X 0,Y 551.918,Z 623.807,A -85,B 0,C 180,E1 25743.115,E2 25743.115} C_VEL
LIN {X 0,Y 551.915,Z 626.043,A -85,B 0,C 180,E1 25741.245,E2 25741.245} C_VEL
LIN {X 0,Y 551.917,Z 626.396,A -85,B 0,C 180,E1 25739.377,E2 25739.377} C_VEL
LIN {X 0,Y 551.911,Z 625.015,A -85,B 0,C 180,E1 25737.612,E2 25737.612} C_VEL
LIN {X 0,Y 551.919,Z 621.948,A -85,B 0,C 180,E1 25735.844,E2 25735.844} C_VEL
LIN {X 0,Y 551.948,Z 616.718,A -85,B 0,C 180,E1 25733.969,E2 25733.969} C_VEL
LIN {X 0,Y 552.017,Z 609.742,A -85,B 0,C 180,E1 25732.192,E2 25732.192} C_VEL
LIN {X 0,Y 552.119,Z 601.742,A -85,B 0,C 180,E1 25730.619,E2 25730.619} C_VEL
LIN {X 0,Y 552.289,Z 591.696,A -85,B 0,C 180,E1 25729.042,E2 25729.042} C_VEL
LIN {X 0,Y 552.523,Z 580.02,A -85,B 0,C 180,E1 25727.564,E2 25727.564} C_VEL
LIN {X 0,Y 552.799,Z 567.132,A -85,B 0,C 180,E1 25726.237,E2 25726.237} C_VEL
LIN {X 0,Y 553.114,Z 553.293,A -85,B 0,C 180,E1 25725.072,E2 25725.072} C_VEL
LIN {X 0,Y 553.446,Z 538.468,A -85,B 0,C 180,E1 25724.061,E2 25724.061} C_VEL
LIN {X 0,Y 553.755,Z 522.568,A -85,B 0,C 180,E1 25723.208,E2 25723.208} C_VEL
LIN {X 0,Y 554.035,Z 506.986,A -85,B 0,C 180,E1 25722.567,E2 25722.567} C_VEL
LIN {X 0,Y 554.259,Z 490.143,A -85,B 0,C 180,E1 25722.073,E2 25722.073} C_VEL
LIN {X 0,Y 554.412,Z 470.925,A -85,B 0,C 180,E1 25721.728,E2 25721.728} C_VEL
LIN {X 0,Y 554.447,Z 456.358,A -85,B 0,C 180,E1 25721.537,E2 25721.537} C_VEL
LIN {X 0,Y 553.539,Z 448.749,A -85,B 0,C 180,E1 25721.408,E2 25721.408} C_VEL
LIN {X 0,Y 547.607,Z 428.809,A -85,B 0,C 180,E1 25720.958,E2 25720.958} C_VEL
LIN {X 0,Y 546.886,Z 422.271,A -85,B 0,C 180,E1 25720.847,E2 25720.847} C_VEL
LIN {X 0,Y 547.171,Z 319.48,A -85,B 0,C 180,E1 25719.442,E2 25719.442} C_VEL
LIN {X 0,Y 546.412,Z 314.503,A -85,B 0,C 180,E1 25719.319,E2 25719.319} C_VEL
LIN {X 0,Y 547.013,Z 281.172,A -85,B 0,C 180,E1 25716.288,E2 25716.288} C_VEL
LIN {X 0,Y 547.51,Z 244.167,A -85,B 0,C 180,E1 25712.952,E2 25712.952} C_VEL
LIN {X 0,Y 547.811,Z 212.391,A -85,B 0,C 180,E1 25710.108,E2 25710.108} C_VEL
LIN {X 0,Y 547.733,Z 185.322,A -85,B 0,C 180,E1 25707.692,E2 25707.692} C_VEL
LIN {X 0,Y 544.402,Z 173.926,A -85,B 0,C 180,E1 25706.473,E2 25706.473} C_VEL
LIN {X 0,Y 544.411,Z 174.03,A -85,B 0,C 180,E1 25703.383,E2 25703.383} C_VEL
LIN {X 0,Y 545.732,Z 177.439,A -85,B 0,C 180,E1 25703.226,E2 25703.226} C_VEL
LIN {X 0,Y 547.468,Z 180.044,A -85,B 0,C 180,E1 25703.051,E2 25703.051} C_VEL
LIN {X 0,Y 554.456,Z 191.807,A -85,B 0,C 180,E1 25702.343,E2 25702.343} C_VEL
LIN {X 0,Y 552.608,Z 415.068,A -85,B 0,C 180,E1 25699.058,E2 25699.058} C_VEL
LIN {X 0,Y 552.173,Z 464.073,A -85,B 0,C 180,E1 25698.312,E2 25698.312} C_VEL
LIN {X 0,Y 551.646,Z 485.605,A -85,B 0,C 180,E1 25697.791,E2 25697.791} C_VEL
LIN {X 0,Y 551.022,Z 507.044,A -85,B 0,C 180,E1 25697.077,E2 25697.077} C_VEL
LIN {X 0,Y 550.321,Z 527.777,A -85,B 0,C 180,E1 25696.193,E2 25696.193} C_VEL
LIN {X 0,Y 549.461,Z 548.522,A -85,B 0,C 180,E1 25695.085,E2 25695.085} C_VEL
LIN {X 0,Y 548.617,Z 568.505,A -85,B 0,C 180,E1 25693.803,E2 25693.803} C_VEL
LIN {X 0,Y 547.716,Z 587.815,A -85,B 0,C 180,E1 25692.325,E2 25692.325} C_VEL
LIN {X 0,Y 546.966,Z 604.713,A -85,B 0,C 180,E1 25690.817,E2 25690.817} C_VEL
LIN {X 0,Y 546.208,Z 621.928,A -85,B 0,C 180,E1 25689.029,E2 25689.029} C_VEL
LIN {X 0,Y 545.573,Z 636.945,A -85,B 0,C 180,E1 25687.214,E2 25687.214} C_VEL
LIN {X 0,Y 545.009,Z 651.961,A -85,B 0,C 180,E1 25685.092,E2 25685.092} C_VEL
LIN {X 0,Y 544.621,Z 663.713,A -85,B 0,C 180,E1 25683.158,E2 25683.158} C_VEL
LIN {X 0,Y 544.311,Z 675.183,A -85,B 0,C 180,E1 25680.924,E2 25680.924} C_VEL
LIN {X 0,Y 544.115,Z 684.306,A -85,B 0,C 180,E1 25678.773,E2 25678.773} C_VEL
LIN {X 0,Y 544.002,Z 692.232,A -85,B 0,C 180,E1 25676.479,E2 25676.479} C_VEL
LIN {X 0,Y 543.947,Z 698.137,A -85,B 0,C 180,E1 25674.254,E2 25674.254} C_VEL
LIN {X 0,Y 543.918,Z 702.646,A -85,B 0,C 180,E1 25671.911,E2 25671.911} C_VEL
LIN {X 0,Y 543.902,Z 705.337,A -85,B 0,C 180,E1 25669.659,E2 25669.659} C_VEL
LIN {X 0,Y 543.901,Z 706.382,A -85,B 0,C 180,E1 25667.547,E2 25667.547} C_VEL
LIN {X 0,Y 543.909,Z 705.972,A -85,B 0,C 180,E1 25665.18,E2 25665.18} C_VEL
LIN {X 0,Y 543.912,Z 703.993,A -85,B 0,C 180,E1 25662.96,E2 25662.96} C_VEL
LIN {X 0,Y 543.918,Z 700.363,A -85,B 0,C 180,E1 25660.7,E2 25660.7} C_VEL
LIN {X 0,Y 543.959,Z 694.847,A -85,B 0,C 180,E1 25658.35,E2 25658.35} C_VEL
LIN {X 0,Y 544.044,Z 688.637,A -85,B 0,C 180,E1 25656.331,E2 25656.331} C_VEL
LIN {X 0,Y 544.2,Z 680.158,A -85,B 0,C 180,E1 25654.109,E2 25654.109} C_VEL
LIN {X 0,Y 544.429,Z 670.363,A -85,B 0,C 180,E1 25652,E2 25652} C_VEL
LIN {X 0,Y 544.753,Z 659.354,A -85,B 0,C 180,E1 25650,E2 25650} C_VEL
LIN {X 0,Y 545.23,Z 645.745,A -85,B 0,C 180,E1 25647.898,E2 25647.898} C_VEL
LIN {X 0,Y 545.802,Z 631.543,A -85,B 0,C 180,E1 25646.008,E2 25646.008} C_VEL
LIN {X 0,Y 546.507,Z 614.914,A -85,B 0,C 180,E1 25644.12,E2 25644.12} C_VEL
LIN {X 0,Y 547.216,Z 598.846,A -85,B 0,C 180,E1 25642.546,E2 25642.546} C_VEL
LIN {X 0,Y 548.11,Z 579.553,A -85,B 0,C 180,E1 25640.921,E2 25640.921} C_VEL
LIN {X 0,Y 548.971,Z 560.416,A -85,B 0,C 180,E1 25639.559,E2 25639.559} C_VEL
LIN {X 0,Y 549.841,Z 539.236,A -85,B 0,C 180,E1 25638.302,E2 25638.302} C_VEL
LIN {X 0,Y 550.531,Z 521.001,A -85,B 0,C 180,E1 25637.412,E2 25637.412} C_VEL
LIN {X 0,Y 551.252,Z 500.51,A -85,B 0,C 180,E1 25636.589,E2 25636.589} C_VEL
LIN {X 0,Y 551.842,Z 478.849,A -85,B 0,C 180,E1 25635.936,E2 25635.936} C_VEL
LIN {X 0,Y 552.247,Z 456.67,A -85,B 0,C 180,E1 25635.468,E2 25635.468} C_VEL
LIN {X 0,Y 553.881,Z 250.601,A -85,B 0,C 180,E1 25632.436,E2 25632.436} C_VEL
LIN {X 0,Y 554.308,Z 191.191,A -85,B 0,C 180,E1 25631.546,E2 25631.546} C_VEL
LIN {X 0,Y 546.266,Z 178.156,A -85,B 0,C 180,E1 25630.737,E2 25630.737} C_VEL
LIN {X 0,Y 544.561,Z 174.911,A -85,B 0,C 180,E1 25630.553,E2 25630.553} C_VEL
LIN {X 0,Y 544.373,Z 173.925,A -85,B 0,C 180,E1 25630.52,E2 25630.52} C_VEL
LIN {X 0,Y 544.4,Z 173.922,A -85,B 0,C 180,E1 25627.199,E2 25627.199} C_VEL
LIN {X 0,Y 544.396,Z 173.921,A -85,B 0,C 180,E1 25623.728,E2 25623.728} C_VEL
LIN {X 0,Y 544.405,Z 173.92,A -85,B 0,C 180,E1 25620.311,E2 25620.311} C_VEL
LIN {X 0,Y 544.39,Z 173.922,A -85,B 0,C 180,E1 25616.942,E2 25616.942} C_VEL
LIN {X 0,Y 544.338,Z 173.927,A -85,B 0,C 180,E1 25613.609,E2 25613.609} C_VEL
LIN {X 0,Y 544.359,Z 173.925,A -85,B 0,C 180,E1 25610.131,E2 25610.131} C_VEL
LIN {X 0,Y 544.402,Z 173.92,A -85,B 0,C 180,E1 25606.815,E2 25606.815} C_VEL
LIN {X 0,Y 544.39,Z 173.923,A -85,B 0,C 180,E1 25603.387,E2 25603.387} C_VEL
LIN {X 0,Y 544.397,Z 173.92,A -85,B 0,C 180,E1 25600.003,E2 25600.003} C_VEL
LIN {X 0,Y 544.403,Z 173.918,A -85,B 0,C 180,E1 25596.621,E2 25596.621} C_VEL
LIN {X 0,Y 544.346,Z 173.927,A -85,B 0,C 180,E1 25593.306,E2 25593.306} C_VEL
LIN {X 0,Y 544.357,Z 173.925,A -85,B 0,C 180,E1 25589.974,E2 25589.974} C_VEL
LIN {X 0,Y 544.404,Z 173.918,A -85,B 0,C 180,E1 25586.742,E2 25586.742} C_VEL
LIN {X 0,Y 544.393,Z 173.916,A -85,B 0,C 180,E1 25583.318,E2 25583.318} C_VEL
LIN {X 0,Y 544.398,Z 173.924,A -85,B 0,C 180,E1 25579.889,E2 25579.889} C_VEL
LIN {X 0,Y 544.405,Z 173.921,A -85,B 0,C 180,E1 25576.43,E2 25576.43} C_VEL
LIN {X 0,Y 544.345,Z 173.92,A -85,B 0,C 180,E1 25573.166,E2 25573.166} C_VEL
LIN {X 0,Y 544.352,Z 173.923,A -85,B 0,C 180,E1 25569.836,E2 25569.836} C_VEL
LIN {X 0,Y 544.404,Z 173.92,A -85,B 0,C 180,E1 25566.539,E2 25566.539} C_VEL
LIN {X 0,Y 544.394,Z 173.924,A -85,B 0,C 180,E1 25563.159,E2 25563.159} C_VEL
LIN {X 0,Y 544.401,Z 173.919,A -85,B 0,C 180,E1 25559.79,E2 25559.79} C_VEL
LIN {X 0,Y 544.403,Z 173.922,A -85,B 0,C 180,E1 25556.42,E2 25556.42} C_VEL
LIN {X 0,Y 544.339,Z 173.927,A -85,B 0,C 180,E1 25553.143,E2 25553.143} C_VEL
LIN {X 0,Y 544.35,Z 173.926,A -85,B 0,C 180,E1 25549.737,E2 25549.737} C_VEL
LIN {X 0,Y 544.404,Z 173.92,A -85,B 0,C 180,E1 25546.404,E2 25546.404} C_VEL
LIN {X 0,Y 544.396,Z 173.923,A -85,B 0,C 180,E1 25543.021,E2 25543.021} C_VEL
LIN {X 0,Y 544.399,Z 173.922,A -85,B 0,C 180,E1 25539.577,E2 25539.577} C_VEL
LIN {X 0,Y 544.407,Z 173.92,A -85,B 0,C 180,E1 25536.153,E2 25536.153} C_VEL
LIN {X 0,Y 544.347,Z 173.924,A -85,B 0,C 180,E1 25532.901,E2 25532.901} C_VEL
LIN {X 0,Y 544.347,Z 173.929,A -85,B 0,C 180,E1 25529.539,E2 25529.539} C_VEL
LIN {X 0,Y 544.413,Z 174.017,A -85,B 0,C 180,E1 25526.818,E2 25526.818} C_VEL
LIN {X 0,Y 545.677,Z 177.359,A -85,B 0,C 180,E1 25526.402,E2 25526.402} C_VEL
LIN {X 0,Y 554.149,Z 194.953,A -85,B 0,C 180,E1 25524.098,E2 25524.098} C_VEL
LIN {X 0,Y 555.898,Z 199.165,A -85,B 0,C 180,E1 25523.591,E2 25523.591} C_VEL
LIN {X 0,Y 554.546,Z 240.303,A -85,B 0,C 180,E1 25520.472,E2 25520.472} C_VEL
LIN {X 0,Y 553.822,Z 274.914,A -85,B 0,C 180,E1 25517.879,E2 25517.879} C_VEL
LIN {X 0,Y 555.323,Z 288.277,A -85,B 0,C 180,E1 25516.758,E2 25516.758} C_VEL
LIN {X 0,Y 558.444,Z 299.222,A -85,B 0,C 180,E1 25515.712,E2 25515.712} C_VEL
LIN {X 0,Y 562.496,Z 307.325,A -85,B 0,C 180,E1 25514.827,E2 25514.827} C_VEL
LIN {X 0,Y 568.022,Z 314.174,A -85,B 0,C 180,E1 25513.951,E2 25513.951} C_VEL
LIN {X 0,Y 575.059,Z 319.669,A -85,B 0,C 180,E1 25513.092,E2 25513.092} C_VEL
LIN {X 0,Y 579.613,Z 321.923,A -85,B 0,C 180,E1 25512.558,E2 25512.558} C_VEL
LIN {X 0,Y 583.179,Z 322.573,A -85,B 0,C 180,E1 25511.963,E2 25511.963} C_VEL
LIN {X 0,Y 585.424,Z 321.839,A -85,B 0,C 180,E1 25511.374,E2 25511.374} C_VEL
LIN {X 0,Y 586.439,Z 319.925,A -85,B 0,C 180,E1 25510.768,E2 25510.768} C_VEL
LIN {X 0,Y 586.073,Z 316.879,A -85,B 0,C 180,E1 25510.189,E2 25510.189} C_VEL
LIN {X 0,Y 584.289,Z 312.863,A -85,B 0,C 180,E1 25509.68,E2 25509.68} C_VEL
LIN {X 0,Y 580.094,Z 306.116,A -85,B 0,C 180,E1 25509.128,E2 25509.128} C_VEL
LIN {X 0,Y 575.392,Z 296.366,A -85,B 0,C 180,E1 25508.549,E2 25508.549} C_VEL
LIN {X 0,Y 571.711,Z 285.36,A -85,B 0,C 180,E1 25508.084,E2 25508.084} C_VEL
LIN {X 0,Y 569.062,Z 273.127,A -85,B 0,C 180,E1 25507.742,E2 25507.742} C_VEL
LIN {X 0,Y 567.43,Z 259.367,A -85,B 0,C 180,E1 25507.529,E2 25507.529} C_VEL
LIN {X 0,Y 566.879,Z 245.236,A -85,B 0,C 180,E1 25507.456,E2 25507.456} C_VEL
LIN {X 0,Y 566.85,Z 218.542,A -85,B 0,C 180,E1 25507.452,E2 25507.452} C_VEL
LIN {X 0,Y 563.373,Z 222.044,A -85,B 0,C 180,E1 25506.988,E2 25506.988} C_VEL
LIN {X 0,Y 561.947,Z 223.011,A -85,B 0,C 180,E1 25506.795,E2 25506.795} C_VEL
LIN {X 0,Y 558.411,Z 231.16,A -85,B 0,C 180,E1 25506.307,E2 25506.307} C_VEL
LIN {X 0,Y 556.53,Z 236.49,A -85,B 0,C 180,E1 25506.042,E2 25506.042} C_VEL
LIN {X 0,Y 555.064,Z 238.243,A -85,B 0,C 180,E1 25505.834,E2 25505.834} C_VEL
LIN {X 0,Y 554.535,Z 238.516,A -85,B 0,C 180,E1 25505.746,E2 25505.746} C_VEL
LIN {X 0,Y 553.062,Z 428.991,A -85,B 0,C 180,E1 25502.919,E2 25502.919} C_VEL
LIN {X 0,Y 552.19,Z 532.732,A -85,B 0,C 180,E1 25501.382,E2 25501.382} C_VEL
LIN {X 0,Y 551.665,Z 555.024,A -85,B 0,C 180,E1 25500.855,E2 25500.855} C_VEL
LIN {X 0,Y 551.037,Z 577.33,A -85,B 0,C 180,E1 25500.113,E2 25500.113} C_VEL
LIN {X 0,Y 550.29,Z 598.565,A -85,B 0,C 180,E1 25499.2,E2 25499.2} C_VEL
LIN {X 0,Y 549.467,Z 618.782,A -85,B 0,C 180,E1 25498.119,E2 25498.119} C_VEL
LIN {X 0,Y 548.592,Z 638.98,A -85,B 0,C 180,E1 25496.814,E2 25496.814} C_VEL
LIN {X 0,Y 547.72,Z 657.948,A -85,B 0,C 180,E1 25495.363,E2 25495.363} C_VEL
LIN {X 0,Y 546.9,Z 676.274,A -85,B 0,C 180,E1 25493.716,E2 25493.716} C_VEL
LIN {X 0,Y 546.12,Z 694.043,A -85,B 0,C 180,E1 25491.839,E2 25491.839} C_VEL
LIN {X 0,Y 545.452,Z 710.286,A -85,B 0,C 180,E1 25489.823,E2 25489.823} C_VEL
LIN {X 0,Y 544.928,Z 724.598,A -85,B 0,C 180,E1 25487.733,E2 25487.733} C_VEL
LIN {X 0,Y 544.525,Z 737.267,A -85,B 0,C 180,E1 25485.55,E2 25485.55} C_VEL
LIN {X 0,Y 544.245,Z 748.313,A -85,B 0,C 180,E1 25483.276,E2 25483.276} C_VEL
LIN {X 0,Y 544.068,Z 757.315,A -85,B 0,C 180,E1 25481.018,E2 25481.018} C_VEL
LIN {X 0,Y 543.967,Z 764.393,A -85,B 0,C 180,E1 25478.775,E2 25478.775} C_VEL
LIN {X 0,Y 543.922,Z 770.007,A -85,B 0,C 180,E1 25476.438,E2 25476.438} C_VEL
LIN {X 0,Y 543.913,Z 773.737,A -85,B 0,C 180,E1 25474.217,E2 25474.217} C_VEL
LIN {X 0,Y 543.908,Z 775.898,A -85,B 0,C 180,E1 25471.896,E2 25471.896} C_VEL
LIN {X 0,Y 543.898,Z 776.439,A -85,B 0,C 180,E1 25469.579,E2 25469.579} C_VEL
LIN {X 0,Y 543.911,Z 775.332,A -85,B 0,C 180,E1 25467.26,E2 25467.26} C_VEL
LIN {X 0,Y 543.923,Z 772.484,A -85,B 0,C 180,E1 25464.938,E2 25464.938} C_VEL
LIN {X 0,Y 543.939,Z 767.932,A -85,B 0,C 180,E1 25462.607,E2 25462.607} C_VEL
LIN {X 0,Y 543.995,Z 761.925,A -85,B 0,C 180,E1 25460.371,E2 25460.371} C_VEL
LIN {X 0,Y 544.118,Z 754.092,A -85,B 0,C 180,E1 25458.123,E2 25458.123} C_VEL
LIN {X 0,Y 544.33,Z 744.349,A -85,B 0,C 180,E1 25455.859,E2 25455.859} C_VEL
LIN {X 0,Y 544.642,Z 733.118,A -85,B 0,C 180,E1 25453.687,E2 25453.687} C_VEL
LIN {X 0,Y 545.069,Z 720.341,A -85,B 0,C 180,E1 25451.608,E2 25451.608} C_VEL
LIN {X 0,Y 545.606,Z 706.039,A -85,B 0,C 180,E1 25449.623,E2 25449.623} C_VEL
LIN {X 0,Y 546.291,Z 689.944,A -85,B 0,C 180,E1 25447.706,E2 25447.706} C_VEL
LIN {X 0,Y 547.06,Z 672.73,A -85,B 0,C 180,E1 25445.947,E2 25445.947} C_VEL
LIN {X 0,Y 547.918,Z 654.039,A -85,B 0,C 180,E1 25444.316,E2 25444.316} C_VEL
LIN {X 0,Y 548.77,Z 634.945,A -85,B 0,C 180,E1 25442.903,E2 25442.903} C_VEL
LIN {X 0,Y 549.636,Z 614.798,A -85,B 0,C 180,E1 25441.654,E2 25441.654} C_VEL
LIN {X 0,Y 550.457,Z 593.657,A -85,B 0,C 180,E1 25440.571,E2 25440.571} C_VEL
LIN {X 0,Y 551.2,Z 572.478,A -85,B 0,C 180,E1 25439.705,E2 25439.705} C_VEL
LIN {X 0,Y 551.794,Z 550.615,A -85,B 0,C 180,E1 25439.024,E2 25439.024} C_VEL
LIN {X 0,Y 552.243,Z 528.602,A -85,B 0,C 180,E1 25438.544,E2 25438.544} C_VEL
LIN {X 0,Y 554.144,Z 297.168,A -85,B 0,C 180,E1 25435.138,E2 25435.138} C_VEL
LIN {X 0,Y 554.772,Z 235.758,A -85,B 0,C 180,E1 25434.208,E2 25434.208} C_VEL
LIN {X 0,Y 556.753,Z 232.774,A -85,B 0,C 180,E1 25433.926,E2 25433.926} C_VEL
LIN {X 0,Y 559.562,Z 224.569,A -85,B 0,C 180,E1 25433.533,E2 25433.533} C_VEL
LIN {X 0,Y 563.638,Z 211.899,A -85,B 0,C 180,E1 25432.976,E2 25432.976} C_VEL
LIN {X 0,Y 564.278,Z 210.308,A -85,B 0,C 180,E1 25432.89,E2 25432.89} C_VEL
LIN {X 0,Y 567.309,Z 206.48,A -85,B 0,C 180,E1 25432.488,E2 25432.488} C_VEL
LIN {X 0,Y 569.293,Z 203.141,A -85,B 0,C 180,E1 25432.228,E2 25432.228} C_VEL
LIN {X 0,Y 583.504,Z 219.463,A -85,B 0,C 180,E1 25430.462,E2 25430.462} C_VEL
LIN {X 0,Y 588.213,Z 223.417,A -85,B 0,C 180,E1 25429.86,E2 25429.86} C_VEL
LIN {X 0,Y 590.537,Z 225.588,A -85,B 0,C 180,E1 25429.318,E2 25429.318} C_VEL
LIN {X 0,Y 591.491,Z 226.917,A -85,B 0,C 180,E1 25428.756,E2 25428.756} C_VEL
LIN {X 0,Y 591.058,Z 227.704,A -85,B 0,C 180,E1 25428.101,E2 25428.101} C_VEL
LIN {X 0,Y 588.88,Z 228.174,A -85,B 0,C 180,E1 25427.467,E2 25427.467} C_VEL
LIN {X 0,Y 585.759,Z 227.462,A -85,B 0,C 180,E1 25426.934,E2 25426.934} C_VEL
LIN {X 0,Y 581.87,Z 225.71,A -85,B 0,C 180,E1 25426.481,E2 25426.481} C_VEL
LIN {X 0,Y 570.977,Z 218.083,A -85,B 0,C 180,E1 25425.313,E2 25425.313} C_VEL
LIN {X 0,Y 565.24,Z 212.818,A -85,B 0,C 180,E1 25424.608,E2 25424.608} C_VEL
LIN {X 0,Y 560.403,Z 206.163,A -85,B 0,C 180,E1 25423.878,E2 25423.878} C_VEL
LIN {X 0,Y 547.954,Z 181.622,A -85,B 0,C 180,E1 25421.481,E2 25421.481} C_VEL
LIN {X 0,Y 546.087,Z 177.919,A -85,B 0,C 180,E1 25421.095,E2 25421.095} C_VEL
LIN {X 0,Y 544.479,Z 174.561,A -85,B 0,C 180,E1 25420.748,E2 25420.748} C_VEL
LIN {X 0,Y 544.369,Z 173.92,A -85,B 0,C 180,E1 25420.661,E2 25420.661} C_VEL
LIN {X 0,Y 544.402,Z 173.92,A -85,B 0,C 180,E1 25417.306,E2 25417.306} C_VEL
LIN {X 0,Y 544.379,Z 173.924,A -85,B 0,C 180,E1 25413.942,E2 25413.942} C_VEL
LIN {X 0,Y 544.407,Z 174.147,A -85,B 0,C 180,E1 25411.961,E2 25411.961} C_VEL
LIN {X 0,Y 545.884,Z 180.487,A -85,B 0,C 180,E1 25411.467,E2 25411.467} C_VEL
LIN {X 0,Y 546.75,Z 212.665,A -85,B 0,C 180,E1 25409.107,E2 25409.107} C_VEL
LIN {X 0,Y 547.175,Z 244.694,A -85,B 0,C 180,E1 25406.595,E2 25406.595} C_VEL
LIN {X 0,Y 547.266,Z 265.415,A -85,B 0,C 180,E1 25404.905,E2 25404.905} C_VEL
LIN {X 0,Y 546.886,Z 301.416,A -85,B 0,C 180,E1 25401.824,E2 25401.824} C_VEL
LIN {X 0,Y 546.726,Z 317.347,A -85,B 0,C 180,E1 25400.468,E2 25400.468} C_VEL
LIN {X 0,Y 547.198,Z 323.294,A -85,B 0,C 180,E1 25400.368,E2 25400.368} C_VEL
LIN {X 0,Y 546.555,Z 484.374,A -85,B 0,C 180,E1 25398.184,E2 25398.184} C_VEL
LIN {X 0,Y 546.412,Z 501.829,A -85,B 0,C 180,E1 25397.75,E2 25397.75} C_VEL
LIN {X 0,Y 546.164,Z 518.544,A -85,B 0,C 180,E1 25397.132,E2 25397.132} C_VEL
LIN {X 0,Y 545.832,Z 534.636,A -85,B 0,C 180,E1 25396.325,E2 25396.325} C_VEL
LIN {X 0,Y 545.468,Z 549.248,A -85,B 0,C 180,E1 25395.382,E2 25395.382} C_VEL
LIN {X 0,Y 545.096,Z 562.887,A -85,B 0,C 180,E1 25394.283,E2 25394.283} C_VEL
LIN {X 0,Y 544.713,Z 576.564,A -85,B 0,C 180,E1 25392.917,E2 25392.917} C_VEL
LIN {X 0,Y 544.419,Z 588.744,A -85,B 0,C 180,E1 25391.44,E2 25391.44} C_VEL
LIN {X 0,Y 544.201,Z 599.379,A -85,B 0,C 180,E1 25389.838,E2 25389.838} C_VEL
LIN {X 0,Y 544.058,Z 607.86,A -85,B 0,C 180,E1 25388.241,E2 25388.241} C_VEL
LIN {X 0,Y 543.975,Z 614.945,A -85,B 0,C 180,E1 25386.543,E2 25386.543} C_VEL
LIN {X 0,Y 543.934,Z 620.482,A -85,B 0,C 180,E1 25384.745,E2 25384.745} C_VEL
LIN {X 0,Y 543.916,Z 624.313,A -85,B 0,C 180,E1 25382.845,E2 25382.845} C_VEL
LIN {X 0,Y 543.913,Z 626.165,A -85,B 0,C 180,E1 25381.053,E2 25381.053} C_VEL
LIN {X 0,Y 543.915,Z 626.375,A -85,B 0,C 180,E1 25379.262,E2 25379.262} C_VEL
LIN {X 0,Y 543.915,Z 624.747,A -85,B 0,C 180,E1 25377.366,E2 25377.366} C_VEL
LIN {X 0,Y 543.926,Z 621.448,A -85,B 0,C 180,E1 25375.572,E2 25375.572} C_VEL
LIN {X 0,Y 543.961,Z 616.368,A -85,B 0,C 180,E1 25373.774,E2 25373.774} C_VEL
LIN {X 0,Y 544.041,Z 609.278,A -85,B 0,C 180,E1 25371.971,E2 25371.971} C_VEL
LIN {X 0,Y 544.18,Z 600.519,A -85,B 0,C 180,E1 25370.268,E2 25370.268} C_VEL
LIN {X 0,Y 544.373,Z 590.809,A -85,B 0,C 180,E1 25368.758,E2 25368.758} C_VEL
LIN {X 0,Y 544.651,Z 579.095,A -85,B 0,C 180,E1 25367.273,E2 25367.273} C_VEL
LIN {X 0,Y 545.031,Z 564.987,A -85,B 0,C 180,E1 25365.823,E2 25365.823} C_VEL
LIN {X 0,Y 545.44,Z 549.963,A -85,B 0,C 180,E1 25364.585,E2 25364.585} C_VEL
LIN {X 0,Y 545.838,Z 534.159,A -85,B 0,C 180,E1 25363.56,E2 25363.56} C_VEL
LIN {X 0,Y 546.16,Z 517.888,A -85,B 0,C 180,E1 25362.748,E2 25362.748} C_VEL
LIN {X 0,Y 546.456,Z 500.858,A -85,B 0,C 180,E1 25362.122,E2 25362.122} C_VEL
LIN {X 0,Y 546.648,Z 483.232,A -85,B 0,C 180,E1 25361.688,E2 25361.688} C_VEL
LIN {X 0,Y 546.886,Z 422.271,A -85,B 0,C 180,E1 25360.847,E2 25360.847} C_VEL
LIN {X 0,Y 545.945,Z 414.667,A -85,B 0,C 180,E1 25360.712,E2 25360.712} C_VEL
LIN {X 0,Y 540.095,Z 394.737,A -85,B 0,C 180,E1 25360.238,E2 25360.238} C_VEL
LIN {X 0,Y 539.448,Z 388.201,A -85,B 0,C 180,E1 25360.124,E2 25360.124} C_VEL
LIN {X 0,Y 539.636,Z 320.59,A -85,B 0,C 180,E1 25359.175,E2 25359.175} C_VEL
LIN {X 0,Y 538.862,Z 315.811,A -85,B 0,C 180,E1 25359.072,E2 25359.072} C_VEL
LIN {X 0,Y 539.518,Z 280.746,A -85,B 0,C 180,E1 25355.88,E2 25355.88} C_VEL
LIN {X 0,Y 540.012,Z 245.236,A -85,B 0,C 180,E1 25352.665,E2 25352.665} C_VEL
LIN {X 0,Y 540.344,Z 210.805,A -85,B 0,C 180,E1 25349.575,E2 25349.575} C_VEL
LIN {X 0,Y 540.394,Z 188.196,A -85,B 0,C 180,E1 25347.534,E2 25347.534} C_VEL
LIN {X 0,Y 536.446,Z 174.915,A -85,B 0,C 180,E1 25346.099,E2 25346.099} C_VEL
LIN {X 0,Y 536.461,Z 175.094,A -85,B 0,C 180,E1 25343.995,E2 25343.995} C_VEL
LIN {X 0,Y 537.76,Z 178.424,A -85,B 0,C 180,E1 25343.836,E2 25343.836} C_VEL
LIN {X 0,Y 539.495,Z 180.877,A -85,B 0,C 180,E1 25343.658,E2 25343.658} C_VEL
LIN {X 0,Y 547.905,Z 194.816,A -85,B 0,C 180,E1 25342.784,E2 25342.784} C_VEL
LIN {X 0,Y 545.808,Z 418.085,A -85,B 0,C 180,E1 25339.461,E2 25339.461} C_VEL
LIN {X 0,Y 545.33,Z 464.289,A -85,B 0,C 180,E1 25338.746,E2 25338.746} C_VEL
LIN {X 0,Y 544.738,Z 485.86,A -85,B 0,C 180,E1 25338.219,E2 25338.219} C_VEL
LIN {X 0,Y 544.018,Z 507.735,A -85,B 0,C 180,E1 25337.477,E2 25337.477} C_VEL
LIN {X 0,Y 543.203,Z 528.736,A -85,B 0,C 180,E1 25336.565,E2 25336.565} C_VEL
LIN {X 0,Y 542.307,Z 547.998,A -85,B 0,C 180,E1 25335.522,E2 25335.522} C_VEL
LIN {X 0,Y 541.329,Z 568.159,A -85,B 0,C 180,E1 25334.221,E2 25334.221} C_VEL
LIN {X 0,Y 540.31,Z 587.548,A -85,B 0,C 180,E1 25332.721,E2 25332.721} C_VEL
LIN {X 0,Y 539.49,Z 603.514,A -85,B 0,C 180,E1 25331.284,E2 25331.284} C_VEL
LIN {X 0,Y 538.586,Z 621.453,A -85,B 0,C 180,E1 25329.413,E2 25329.413} C_VEL
LIN {X 0,Y 537.824,Z 637.087,A -85,B 0,C 180,E1 25327.5,E2 25327.5} C_VEL
LIN {X 0,Y 537.183,Z 651.928,A -85,B 0,C 180,E1 25325.371,E2 25325.371} C_VEL
LIN {X 0,Y 536.751,Z 663.54,A -85,B 0,C 180,E1 25323.432,E2 25323.432} C_VEL
LIN {X 0,Y 536.386,Z 675.008,A -85,B 0,C 180,E1 25321.172,E2 25321.172} C_VEL
LIN {X 0,Y 536.145,Z 684.564,A -85,B 0,C 180,E1 25318.882,E2 25318.882} C_VEL
LIN {X 0,Y 536.014,Z 692.306,A -85,B 0,C 180,E1 25316.596,E2 25316.596} C_VEL
LIN {X 0,Y 535.95,Z 697.966,A -85,B 0,C 180,E1 25314.438,E2 25314.438} C_VEL
LIN {X 0,Y 535.925,Z 702.591,A -85,B 0,C 180,E1 25312.025,E2 25312.025} C_VEL
LIN {X 0,Y 535.902,Z 705.305,A -85,B 0,C 180,E1 25309.737,E2 25309.737} C_VEL
LIN {X 0,Y 535.901,Z 706.382,A -85,B 0,C 180,E1 25307.559,E2 25307.559} C_VEL
LIN {X 0,Y 535.912,Z 705.966,A -85,B 0,C 180,E1 25305.142,E2 25305.142} C_VEL
LIN {X 0,Y 535.912,Z 704.035,A -85,B 0,C 180,E1 25302.938,E2 25302.938} C_VEL
LIN {X 0,Y 535.92,Z 700.438,A -85,B 0,C 180,E1 25300.644,E2 25300.644} C_VEL
LIN {X 0,Y 535.97,Z 694.952,A -85,B 0,C 180,E1 25298.259,E2 25298.259} C_VEL
LIN {X 0,Y 536.067,Z 688.738,A -85,B 0,C 180,E1 25296.202,E2 25296.202} C_VEL
LIN {X 0,Y 536.262,Z 679.88,A -85,B 0,C 180,E1 25293.849,E2 25293.849} C_VEL
LIN {X 0,Y 536.533,Z 670.03,A -85,B 0,C 180,E1 25291.709,E2 25291.709} C_VEL
LIN {X 0,Y 536.932,Z 658.369,A -85,B 0,C 180,E1 25289.573,E2 25289.573} C_VEL
LIN {X 0,Y 537.46,Z 645.305,A -85,B 0,C 180,E1 25287.548,E2 25287.548} C_VEL
LIN {X 0,Y 538.126,Z 631.042,A -85,B 0,C 180,E1 25285.631,E2 25285.631} C_VEL
LIN {X 0,Y 538.94,Z 614.305,A -85,B 0,C 180,E1 25283.716,E2 25283.716} C_VEL
LIN {X 0,Y 539.76,Z 598.171,A -85,B 0,C 180,E1 25282.121,E2 25282.121} C_VEL
LIN {X 0,Y 540.775,Z 578.725,A -85,B 0,C 180,E1 25280.475,E2 25280.475} C_VEL
LIN {X 0,Y 541.778,Z 559.438,A -85,B 0,C 180,E1 25279.096,E2 25279.096} C_VEL
LIN {X 0,Y 542.718,Z 538.976,A -85,B 0,C 180,E1 25277.876,E2 25277.876} C_VEL
LIN {X 0,Y 543.504,Z 520.681,A -85,B 0,C 180,E1 25276.976,E2 25276.976} C_VEL
LIN {X 0,Y 544.308,Z 500.073,A -85,B 0,C 180,E1 25276.144,E2 25276.144} C_VEL
LIN {X 0,Y 544.972,Z 478.604,A -85,B 0,C 180,E1 25275.493,E2 25275.493} C_VEL
LIN {X 0,Y 545.421,Z 456.612,A -85,B 0,C 180,E1 25275.026,E2 25275.026} C_VEL
LIN {X 0,Y 547.274,Z 252.258,A -85,B 0,C 180,E1 25271.985,E2 25271.985} C_VEL
LIN {X 0,Y 547.724,Z 194.417,A -85,B 0,C 180,E1 25271.106,E2 25271.106} C_VEL
LIN {X 0,Y 538.445,Z 179.311,A -85,B 0,C 180,E1 25270.143,E2 25270.143} C_VEL
LIN {X 0,Y 536.657,Z 176.065,A -85,B 0,C 180,E1 25269.947,E2 25269.947} C_VEL
LIN {X 0,Y 536.429,Z 174.915,A -85,B 0,C 180,E1 25269.886,E2 25269.886} C_VEL
LIN {X 0,Y 536.447,Z 174.91,A -85,B 0,C 180,E1 25266.493,E2 25266.493} C_VEL
LIN {X 0,Y 536.45,Z 174.91,A -85,B 0,C 180,E1 25263.189,E2 25263.189} C_VEL
LIN {X 0,Y 536.432,Z 174.915,A -85,B 0,C 180,E1 25259.785,E2 25259.785} C_VEL
LIN {X 0,Y 536.444,Z 174.914,A -85,B 0,C 180,E1 25256.424,E2 25256.424} C_VEL
LIN {X 0,Y 536.456,Z 174.912,A -85,B 0,C 180,E1 25252.913,E2 25252.913} C_VEL
LIN {X 0,Y 536.436,Z 174.916,A -85,B 0,C 180,E1 25249.561,E2 25249.561} C_VEL
LIN {X 0,Y 536.444,Z 174.912,A -85,B 0,C 180,E1 25246.164,E2 25246.164} C_VEL
LIN {X 0,Y 536.463,Z 174.908,A -85,B 0,C 180,E1 25242.721,E2 25242.721} C_VEL
LIN {X 0,Y 536.429,Z 174.912,A -85,B 0,C 180,E1 25239.465,E2 25239.465} C_VEL
LIN {X 0,Y 536.426,Z 174.912,A -85,B 0,C 180,E1 25236.087,E2 25236.087} C_VEL
LIN {X 0,Y 536.46,Z 174.907,A -85,B 0,C 180,E1 25232.718,E2 25232.718} C_VEL
LIN {X 0,Y 536.441,Z 174.915,A -85,B 0,C 180,E1 25229.354,E2 25229.354} C_VEL
LIN {X 0,Y 536.439,Z 174.91,A -85,B 0,C 180,E1 25225.978,E2 25225.978} C_VEL
LIN {X 0,Y 536.466,Z 174.899,A -85,B 0,C 180,E1 25222.578,E2 25222.578} C_VEL
LIN {X 0,Y 536.432,Z 174.909,A -85,B 0,C 180,E1 25219.264,E2 25219.264} C_VEL
LIN {X 0,Y 536.425,Z 174.916,A -85,B 0,C 180,E1 25215.89,E2 25215.89} C_VEL
LIN {X 0,Y 536.453,Z 174.908,A -85,B 0,C 180,E1 25212.596,E2 25212.596} C_VEL
LIN {X 0,Y 536.436,Z 174.912,A -85,B 0,C 180,E1 25209.224,E2 25209.224} C_VEL
LIN {X 0,Y 536.437,Z 174.912,A -85,B 0,C 180,E1 25205.884,E2 25205.884} C_VEL
LIN {X 0,Y 536.462,Z 174.908,A -85,B 0,C 180,E1 25202.457,E2 25202.457} C_VEL
LIN {X 0,Y 536.434,Z 174.91,A -85,B 0,C 180,E1 25199.146,E2 25199.146} C_VEL
LIN {X 0,Y 536.425,Z 174.91,A -85,B 0,C 180,E1 25195.714,E2 25195.714} C_VEL
LIN {X 0,Y 536.454,Z 174.908,A -85,B 0,C 180,E1 25192.396,E2 25192.396} C_VEL
LIN {X 0,Y 536.437,Z 174.915,A -85,B 0,C 180,E1 25189.041,E2 25189.041} C_VEL
LIN {X 0,Y 536.437,Z 174.913,A -85,B 0,C 180,E1 25185.647,E2 25185.647} C_VEL
LIN {X 0,Y 536.458,Z 174.908,A -85,B 0,C 180,E1 25182.202,E2 25182.202} C_VEL
LIN {X 0,Y 536.438,Z 174.906,A -85,B 0,C 180,E1 25178.917,E2 25178.917} C_VEL
LIN {X 0,Y 536.42,Z 174.915,A -85,B 0,C 180,E1 25175.451,E2 25175.451} C_VEL
LIN {X 0,Y 536.452,Z 174.916,A -85,B 0,C 180,E1 25172.228,E2 25172.228} C_VEL
LIN {X 0,Y 536.434,Z 174.912,A -85,B 0,C 180,E1 25168.916,E2 25168.916} C_VEL
LIN {X 0,Y 536.44,Z 175.069,A -85,B 0,C 180,E1 25167.582,E2 25167.582} C_VEL
LIN {X 0,Y 537.872,Z 178.586,A -85,B 0,C 180,E1 25167.126,E2 25167.126} C_VEL
LIN {X 0,Y 544.775,Z 192.909,A -85,B 0,C 180,E1 25165.195,E2 25165.195} C_VEL
LIN {X 0,Y 549.414,Z 203.05,A -85,B 0,C 180,E1 25163.903,E2 25163.903} C_VEL
LIN {X 0,Y 547.835,Z 245.805,A -85,B 0,C 180,E1 25160.638,E2 25160.638} C_VEL
LIN {X 0,Y 547.106,Z 277.846,A -85,B 0,C 180,E1 25158.214,E2 25158.214} C_VEL
LIN {X 0,Y 548.483,Z 291.038,A -85,B 0,C 180,E1 25157.096,E2 25157.096} C_VEL
LIN {X 0,Y 551.466,Z 302.276,A -85,B 0,C 180,E1 25156.02,E2 25156.02} C_VEL
LIN {X 0,Y 555.826,Z 311.522,A -85,B 0,C 180,E1 25155.013,E2 25155.013} C_VEL
LIN {X 0,Y 561.8,Z 319.252,A -85,B 0,C 180,E1 25154.027,E2 25154.027} C_VEL
LIN {X 0,Y 568.725,Z 325.002,A -85,B 0,C 180,E1 25153.148,E2 25153.148} C_VEL
LIN {X 0,Y 575.555,Z 328.66,A -85,B 0,C 180,E1 25152.412,E2 25152.412} C_VEL
LIN {X 0,Y 579.097,Z 329.557,A -85,B 0,C 180,E1 25151.914,E2 25151.914} C_VEL
LIN {X 0,Y 581.909,Z 329.277,A -85,B 0,C 180,E1 25151.335,E2 25151.335} C_VEL
LIN {X 0,Y 583.489,Z 327.904,A -85,B 0,C 180,E1 25150.759,E2 25150.759} C_VEL
LIN {X 0,Y 583.822,Z 325.335,A -85,B 0,C 180,E1 25150.15,E2 25150.15} C_VEL
LIN {X 0,Y 582.692,Z 321.8,A -85,B 0,C 180,E1 25149.597,E2 25149.597} C_VEL
LIN {X 0,Y 580.171,Z 317.48,A -85,B 0,C 180,E1 25149.138,E2 25149.138} C_VEL
LIN {X 0,Y 574.691,Z 308.368,A -85,B 0,C 180,E1 25148.461,E2 25148.461} C_VEL
LIN {X 0,Y 570.134,Z 297.818,A -85,B 0,C 180,E1 25147.881,E2 25147.881} C_VEL
LIN {X 0,Y 566.509,Z 285.793,A -85,B 0,C 180,E1 25147.407,E2 25147.407} C_VEL
LIN {X 0,Y 563.975,Z 272.685,A -85,B 0,C 180,E1 25147.069,E2 25147.069} C_VEL
LIN {X 0,Y 562.481,Z 258.183,A -85,B 0,C 180,E1 25146.867,E2 25146.867} C_VEL
LIN {X 0,Y 562.048,Z 243.214,A -85,B 0,C 180,E1 25146.808,E2 25146.808} C_VEL
LIN {X 0,Y 561.985,Z 237.124,A -85,B 0,C 180,E1 25146.8,E2 25146.8} C_VEL
LIN {X 0,Y 559.709,Z 242.452,A -85,B 0,C 180,E1 25146.487,E2 25146.487} C_VEL
LIN {X 0,Y 558.8,Z 244.184,A -85,B 0,C 180,E1 25146.361,E2 25146.361} C_VEL
LIN {X 0,Y 554.551,Z 293,A -85,B 0,C 180,E1 25145.76,E2 25145.76} C_VEL
LIN {X 0,Y 550.923,Z 324.674,A -85,B 0,C 180,E1 25145.233,E2 25145.233} C_VEL
LIN {X 0,Y 548.625,Z 338.357,A -85,B 0,C 180,E1 25144.892,E2 25144.892} C_VEL
LIN {X 0,Y 547.556,Z 341.648,A -85,B 0,C 180,E1 25144.731,E2 25144.731} C_VEL
LIN {X 0,Y 547.155,Z 342.215,A -85,B 0,C 180,E1 25144.666,E2 25144.666} C_VEL
LIN {X 0,Y 545.364,Z 532.367,A -85,B 0,C 180,E1 25141.829,E2 25141.829} C_VEL
LIN {X 0,Y 544.783,Z 554.52,A -85,B 0,C 180,E1 25141.303,E2 25141.303} C_VEL
LIN {X 0,Y 544.06,Z 577.325,A -85,B 0,C 180,E1 25140.54,E2 25140.54} C_VEL
LIN {X 0,Y 543.205,Z 598.56,A -85,B 0,C 180,E1 25139.618,E2 25139.618} C_VEL
LIN {X 0,Y 542.289,Z 618.789,A -85,B 0,C 180,E1 25138.525,E2 25138.525} C_VEL
LIN {X 0,Y 541.287,Z 638.985,A -85,B 0,C 180,E1 25137.205,E2 25137.205} C_VEL
LIN {X 0,Y 540.25,Z 658.826,A -85,B 0,C 180,E1 25135.663,E2 25135.663} C_VEL
LIN {X 0,Y 539.33,Z 676.834,A -85,B 0,C 180,E1 25134.012,E2 25134.012} C_VEL
LIN {X 0,Y 538.461,Z 694.223,A -85,B 0,C 180,E1 25132.145,E2 25132.145} C_VEL
LIN {X 0,Y 537.697,Z 710.397,A -85,B 0,C 180,E1 25130.107,E2 25130.107} C_VEL
LIN {X 0,Y 537.082,Z 724.891,A -85,B 0,C 180,E1 25127.955,E2 25127.955} C_VEL
LIN {X 0,Y 536.622,Z 737.271,A -85,B 0,C 180,E1 25125.785,E2 25125.785} C_VEL
LIN {X 0,Y 536.303,Z 748.316,A -85,B 0,C 180,E1 25123.476,E2 25123.476} C_VEL
LIN {X 0,Y 536.099,Z 757.325,A -85,B 0,C 180,E1 25121.181,E2 25121.181} C_VEL
LIN {X 0,Y 535.984,Z 764.396,A -85,B 0,C 180,E1 25118.907,E2 25118.907} C_VEL
LIN {X 0,Y 535.927,Z 770.01,A -85,B 0,C 180,E1 25116.535,E2 25116.535} C_VEL
LIN {X 0,Y 535.914,Z 773.738,A -85,B 0,C 180,E1 25114.28,E2 25114.28} C_VEL
LIN {X 0,Y 535.909,Z 775.9,A -85,B 0,C 180,E1 25111.924,E2 25111.924} C_VEL
LIN {X 0,Y 535.898,Z 776.442,A -85,B 0,C 180,E1 25109.572,E2 25109.572} C_VEL
LIN {X 0,Y 535.912,Z 775.331,A -85,B 0,C 180,E1 25107.219,E2 25107.219} C_VEL
LIN {X 0,Y 535.923,Z 772.486,A -85,B 0,C 180,E1 25104.862,E2 25104.862} C_VEL
LIN {X 0,Y 535.945,Z 767.936,A -85,B 0,C 180,E1 25102.496,E2 25102.496} C_VEL
LIN {X 0,Y 536.012,Z 761.924,A -85,B 0,C 180,E1 25100.227,E2 25100.227} C_VEL
LIN {X 0,Y 536.158,Z 754.096,A -85,B 0,C 180,E1 25097.944,E2 25097.944} C_VEL
LIN {X 0,Y 536.406,Z 744.352,A -85,B 0,C 180,E1 25095.646,E2 25095.646} C_VEL
LIN {X 0,Y 536.771,Z 733.119,A -85,B 0,C 180,E1 25093.441,E2 25093.441} C_VEL
LIN {X 0,Y 537.294,Z 719.627,A -85,B 0,C 180,E1 25091.22,E2 25091.22} C_VEL
LIN {X 0,Y 537.914,Z 705.192,A -85,B 0,C 180,E1 25089.205,E2 25089.205} C_VEL
LIN {X 0,Y 538.69,Z 689.207,A -85,B 0,C 180,E1 25087.29,E2 25087.29} C_VEL
LIN {X 0,Y 539.599,Z 671.529,A -85,B 0,C 180,E1 25085.476,E2 25085.476} C_VEL
LIN {X 0,Y 540.557,Z 653.315,A -85,B 0,C 180,E1 25083.882,E2 25083.882} C_VEL
LIN {X 0,Y 541.536,Z 633.999,A -85,B 0,C 180,E1 25082.445,E2 25082.445} C_VEL
LIN {X 0,Y 542.516,Z 613.784,A -85,B 0,C 180,E1 25081.187,E2 25081.187} C_VEL
LIN {X 0,Y 543.469,Z 592.406,A -85,B 0,C 180,E1 25080.094,E2 25080.094} C_VEL
LIN {X 0,Y 544.284,Z 570.863,A -85,B 0,C 180,E1 25079.217,E2 25079.217} C_VEL
LIN {X 0,Y 544.977,Z 548.714,A -85,B 0,C 180,E1 25078.539,E2 25078.539} C_VEL
LIN {X 0,Y 545.436,Z 526.682,A -85,B 0,C 180,E1 25078.071,E2 25078.071} C_VEL
LIN {X 0,Y 547.272,Z 342.149,A -85,B 0,C 180,E1 25075.312,E2 25075.312} C_VEL
LIN {X 0,Y 548.27,Z 339.897,A -85,B 0,C 180,E1 25075.161,E2 25075.161} C_VEL
LIN {X 0,Y 550.348,Z 328.651,A -85,B 0,C 180,E1 25074.852,E2 25074.852} C_VEL
LIN {X 0,Y 553.858,Z 299.649,A -85,B 0,C 180,E1 25074.339,E2 25074.339} C_VEL
LIN {X 0,Y 558.053,Z 253.746,A -85,B 0,C 180,E1 25073.743,E2 25073.743} C_VEL
LIN {X 0,Y 559.265,Z 240.022,A -85,B 0,C 180,E1 25073.574,E2 25073.574} C_VEL
LIN {X 0,Y 561.5,Z 235.067,A -85,B 0,C 180,E1 25073.266,E2 25073.266} C_VEL
LIN {X 0,Y 563.826,Z 228.273,A -85,B 0,C 180,E1 25072.951,E2 25072.951} C_VEL
LIN {X 0,Y 567.918,Z 216.036,A -85,B 0,C 180,E1 25072.407,E2 25072.407} C_VEL
LIN {X 0,Y 569.753,Z 213.705,A -85,B 0,C 180,E1 25072.168,E2 25072.168} C_VEL
LIN {X 0,Y 581.123,Z 226.541,A -85,B 0,C 180,E1 25070.747,E2 25070.747} C_VEL
LIN {X 0,Y 586.282,Z 230.836,A -85,B 0,C 180,E1 25070.084,E2 25070.084} C_VEL
LIN {X 0,Y 588.579,Z 233.019,A -85,B 0,C 180,E1 25069.539,E2 25069.539} C_VEL
LIN {X 0,Y 589.493,Z 234.409,A -85,B 0,C 180,E1 25068.973,E2 25068.973} C_VEL
LIN {X 0,Y 588.952,Z 235.2,A -85,B 0,C 180,E1 25068.279,E2 25068.279} C_VEL
LIN {X 0,Y 586.82,Z 235.686,A -85,B 0,C 180,E1 25067.686,E2 25067.686} C_VEL
LIN {X 0,Y 583.417,Z 235.034,A -85,B 0,C 180,E1 25067.126,E2 25067.126} C_VEL
LIN {X 0,Y 578.959,Z 233.183,A -85,B 0,C 180,E1 25066.64,E2 25066.64} C_VEL
LIN {X 0,Y 571.26,Z 228.252,A -85,B 0,C 180,E1 25065.844,E2 25065.844} C_VEL
LIN {X 0,Y 562.081,Z 220.969,A -85,B 0,C 180,E1 25064.783,E2 25064.783} C_VEL
LIN {X 0,Y 556.162,Z 213.863,A -85,B 0,C 180,E1 25063.943,E2 25063.943} C_VEL
LIN {X 0,Y 547.217,Z 196.564,A -85,B 0,C 180,E1 25062.252,E2 25062.252} C_VEL
LIN {X 0,Y 540.121,Z 182.745,A -85,B 0,C 180,E1 25060.803,E2 25060.803} C_VEL
LIN {X 0,Y 537.991,Z 178.753,A -85,B 0,C 180,E1 25060.36,E2 25060.36} C_VEL
LIN {X 0,Y 536.515,Z 175.377,A -85,B 0,C 180,E1 25060.008,E2 25060.008} C_VEL
LIN {X 0,Y 536.448,Z 174.91,A -85,B 0,C 180,E1 25059.932,E2 25059.932} C_VEL
